// TIA Portal V17 export
// export: Created 2025-03-13T10:29:50.4111857Z, ExportSetting WithDefaults, DisplayName Totally Integrated Automation Portal, DisplayVersion V17 Update 8, DisplayName TIA Portal Openness, DisplayVersion V17 Update 8, DisplayName TIA Portal Version Control Interface, DisplayVersion V17, DisplayName SINAMICS Startdrive Advanced, DisplayVersion V17 SP2, DisplayName SINAMICS Startdrive G110M, G120, G120C, G120D, G120P, G115D, DisplayVersion V17 SP2, DisplayName SINAMICS Startdrive G130, G150, S120, S150, SINAMICS MV, S210, DisplayVersion V17 SP2, DisplayName STEP 7 Professional, DisplayVersion V17 Update 8, DisplayName SINUMERIK ONE STEP 7 Toolbox, DisplayVersion V17 Update 12, DisplayName SINUMERIK 840D sl STEP 7 Toolbox, DisplayVersion V17 Update 12, DisplayName STEP 7 Safety, DisplayVersion V17 Update 6, DisplayName WinCC Advanced, DisplayVersion V17 Update 8
FUNCTION "FC7330_ROBOT_CELL_TO_MACHINE_INTERLOCK" : Void   // FC7330, LAD
{ S7_Optimized_Access := 'FALSE' }
AUTHOR : ETXETAR
VERSION : 1.0
// stored: AutoNumber false, IsIECCheckEnabled false, SetENOAutomatically false, UDAEnableTagReadback false
   VAR_TEMP
      dry_load_side0 : Bool;
      dry_load_side180 : Bool;
      Status_receive : Int;
      QC_FORECAST : Int;
      QC_EXPIRED : Int;
      QC_COUNTS : Int;
      RETVAL_FILL : Int;
      temp0 : Int;
      status_sfc21 : Int;
      RETVAL_FILL_1 : Int;
      ONE : Byte;
      ZERO : Byte;
      retval_sfc21 : Int;
      COUNTS_FOR_ERROR_UNIT_01 : Int;
      COUNTS_FOR_ERROR_UNIT_02 : Int;
      AUX_1_GTRY_SWITCH_OFF : Bool;
      AUX_2_GTRY_SWITCH_OFF : Bool;
      WITH_MANUAL_LOADER : Bool;
      WITH_OUT_MANUAL_LOADER : Bool;
   END_VAR
   VAR CONSTANT
      FC_NUMBER : DInt := 7330;   // FC NUMBER
   END_VAR
   VAR_TEMP   // added for the SCL form of the ladder/FBD networks
      _w1 : Bool;
      _w2 : Bool;
   END_VAR
BEGIN

REGION Network 1: >>>>>>>>>>>>>>>> INTERLOCKS CELL TO MACHINE GENERAL <<<<<<<<<<<<<<<<
END_REGION

REGION Network 2: MEASURING STATION START MEASURING CYCLE
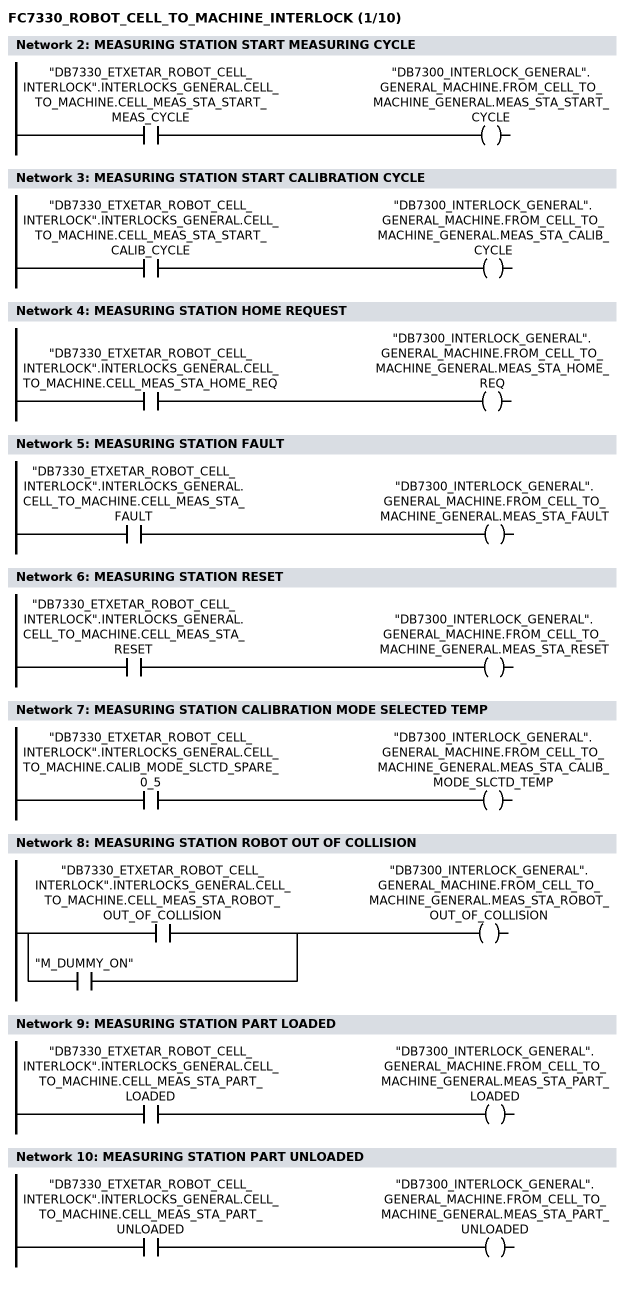
   RUNG wire#powerrail
      Contact( "DB7330_ETXETAR_ROBOT_CELL_INTERLOCK".INTERLOCKS_GENERAL.CELL_TO_MACHINE.CELL_MEAS_STA_START_MEAS_CYCLE )
      Coil( "DB7300_INTERLOCK_GENERAL".GENERAL_MACHINE.FROM_CELL_TO_MACHINE_GENERAL.MEAS_STA_START_CYCLE )
   END_RUNG
   // the same network as SCL:
   "DB7300_INTERLOCK_GENERAL".GENERAL_MACHINE.FROM_CELL_TO_MACHINE_GENERAL.MEAS_STA_START_CYCLE := "DB7330_ETXETAR_ROBOT_CELL_INTERLOCK".INTERLOCKS_GENERAL.CELL_TO_MACHINE.CELL_MEAS_STA_START_MEAS_CYCLE;
END_REGION

REGION Network 3: MEASURING STATION START CALIBRATION CYCLE
   RUNG wire#powerrail
      Contact( "DB7330_ETXETAR_ROBOT_CELL_INTERLOCK".INTERLOCKS_GENERAL.CELL_TO_MACHINE.CELL_MEAS_STA_START_CALIB_CYCLE )
      Coil( "DB7300_INTERLOCK_GENERAL".GENERAL_MACHINE.FROM_CELL_TO_MACHINE_GENERAL.MEAS_STA_CALIB_CYCLE )
   END_RUNG
   // the same network as SCL:
   "DB7300_INTERLOCK_GENERAL".GENERAL_MACHINE.FROM_CELL_TO_MACHINE_GENERAL.MEAS_STA_CALIB_CYCLE := "DB7330_ETXETAR_ROBOT_CELL_INTERLOCK".INTERLOCKS_GENERAL.CELL_TO_MACHINE.CELL_MEAS_STA_START_CALIB_CYCLE;
END_REGION

REGION Network 4: MEASURING STATION HOME REQUEST
   RUNG wire#powerrail
      Contact( "DB7330_ETXETAR_ROBOT_CELL_INTERLOCK".INTERLOCKS_GENERAL.CELL_TO_MACHINE.CELL_MEAS_STA_HOME_REQ )
      Coil( "DB7300_INTERLOCK_GENERAL".GENERAL_MACHINE.FROM_CELL_TO_MACHINE_GENERAL.MEAS_STA_HOME_REQ )
   END_RUNG
   // the same network as SCL:
   "DB7300_INTERLOCK_GENERAL".GENERAL_MACHINE.FROM_CELL_TO_MACHINE_GENERAL.MEAS_STA_HOME_REQ := "DB7330_ETXETAR_ROBOT_CELL_INTERLOCK".INTERLOCKS_GENERAL.CELL_TO_MACHINE.CELL_MEAS_STA_HOME_REQ;
END_REGION

REGION Network 5: MEASURING STATION FAULT
   RUNG wire#powerrail
      Contact( "DB7330_ETXETAR_ROBOT_CELL_INTERLOCK".INTERLOCKS_GENERAL.CELL_TO_MACHINE.CELL_MEAS_STA_FAULT )
      Coil( "DB7300_INTERLOCK_GENERAL".GENERAL_MACHINE.FROM_CELL_TO_MACHINE_GENERAL.MEAS_STA_FAULT )
   END_RUNG
   // the same network as SCL:
   "DB7300_INTERLOCK_GENERAL".GENERAL_MACHINE.FROM_CELL_TO_MACHINE_GENERAL.MEAS_STA_FAULT := "DB7330_ETXETAR_ROBOT_CELL_INTERLOCK".INTERLOCKS_GENERAL.CELL_TO_MACHINE.CELL_MEAS_STA_FAULT;
END_REGION

REGION Network 6: MEASURING STATION RESET
   RUNG wire#powerrail
      Contact( "DB7330_ETXETAR_ROBOT_CELL_INTERLOCK".INTERLOCKS_GENERAL.CELL_TO_MACHINE.CELL_MEAS_STA_RESET )
      Coil( "DB7300_INTERLOCK_GENERAL".GENERAL_MACHINE.FROM_CELL_TO_MACHINE_GENERAL.MEAS_STA_RESET )
   END_RUNG
   // the same network as SCL:
   "DB7300_INTERLOCK_GENERAL".GENERAL_MACHINE.FROM_CELL_TO_MACHINE_GENERAL.MEAS_STA_RESET := "DB7330_ETXETAR_ROBOT_CELL_INTERLOCK".INTERLOCKS_GENERAL.CELL_TO_MACHINE.CELL_MEAS_STA_RESET;
END_REGION

REGION Network 7: MEASURING STATION CALIBRATION MODE SELECTED TEMP
   RUNG wire#powerrail
      Contact( "DB7330_ETXETAR_ROBOT_CELL_INTERLOCK".INTERLOCKS_GENERAL.CELL_TO_MACHINE.CALIB_MODE_SLCTD_SPARE_0_5 )
      Coil( "DB7300_INTERLOCK_GENERAL".GENERAL_MACHINE.FROM_CELL_TO_MACHINE_GENERAL.MEAS_STA_CALIB_MODE_SLCTD_TEMP )
   END_RUNG
   // the same network as SCL:
   "DB7300_INTERLOCK_GENERAL".GENERAL_MACHINE.FROM_CELL_TO_MACHINE_GENERAL.MEAS_STA_CALIB_MODE_SLCTD_TEMP := "DB7330_ETXETAR_ROBOT_CELL_INTERLOCK".INTERLOCKS_GENERAL.CELL_TO_MACHINE.CALIB_MODE_SLCTD_SPARE_0_5;
END_REGION

REGION Network 8: MEASURING STATION ROBOT OUT OF COLLISION
   RUNG wire#powerrail
      Contact( "DB7330_ETXETAR_ROBOT_CELL_INTERLOCK".INTERLOCKS_GENERAL.CELL_TO_MACHINE.CELL_MEAS_STA_ROBOT_OUT_OF_COLLISION )
      wire#w1
      Coil( "DB7300_INTERLOCK_GENERAL".GENERAL_MACHINE.FROM_CELL_TO_MACHINE_GENERAL.MEAS_STA_ROBOT_OUT_OF_COLLISION )
   END_RUNG
   RUNG wire#powerrail
      Contact( "M_DUMMY_ON" )
   END_RUNG wire#w1
   // the same network as SCL:
   "DB7300_INTERLOCK_GENERAL".GENERAL_MACHINE.FROM_CELL_TO_MACHINE_GENERAL.MEAS_STA_ROBOT_OUT_OF_COLLISION := "DB7330_ETXETAR_ROBOT_CELL_INTERLOCK".INTERLOCKS_GENERAL.CELL_TO_MACHINE.CELL_MEAS_STA_ROBOT_OUT_OF_COLLISION OR "M_DUMMY_ON";
END_REGION

REGION Network 9: MEASURING STATION PART LOADED
   RUNG wire#powerrail
      Contact( "DB7330_ETXETAR_ROBOT_CELL_INTERLOCK".INTERLOCKS_GENERAL.CELL_TO_MACHINE.CELL_MEAS_STA_PART_LOADED )
      Coil( "DB7300_INTERLOCK_GENERAL".GENERAL_MACHINE.FROM_CELL_TO_MACHINE_GENERAL.MEAS_STA_PART_LOADED )
   END_RUNG
   // the same network as SCL:
   "DB7300_INTERLOCK_GENERAL".GENERAL_MACHINE.FROM_CELL_TO_MACHINE_GENERAL.MEAS_STA_PART_LOADED := "DB7330_ETXETAR_ROBOT_CELL_INTERLOCK".INTERLOCKS_GENERAL.CELL_TO_MACHINE.CELL_MEAS_STA_PART_LOADED;
END_REGION

REGION Network 10: MEASURING STATION PART UNLOADED
   RUNG wire#powerrail
      Contact( "DB7330_ETXETAR_ROBOT_CELL_INTERLOCK".INTERLOCKS_GENERAL.CELL_TO_MACHINE.CELL_MEAS_STA_PART_UNLOADED )
      Coil( "DB7300_INTERLOCK_GENERAL".GENERAL_MACHINE.FROM_CELL_TO_MACHINE_GENERAL.MEAS_STA_PART_UNLOADED )
   END_RUNG
   // the same network as SCL:
   "DB7300_INTERLOCK_GENERAL".GENERAL_MACHINE.FROM_CELL_TO_MACHINE_GENERAL.MEAS_STA_PART_UNLOADED := "DB7330_ETXETAR_ROBOT_CELL_INTERLOCK".INTERLOCKS_GENERAL.CELL_TO_MACHINE.CELL_MEAS_STA_PART_UNLOADED;
END_REGION

REGION Network 11: CELL COOLING DEGRADED MODE
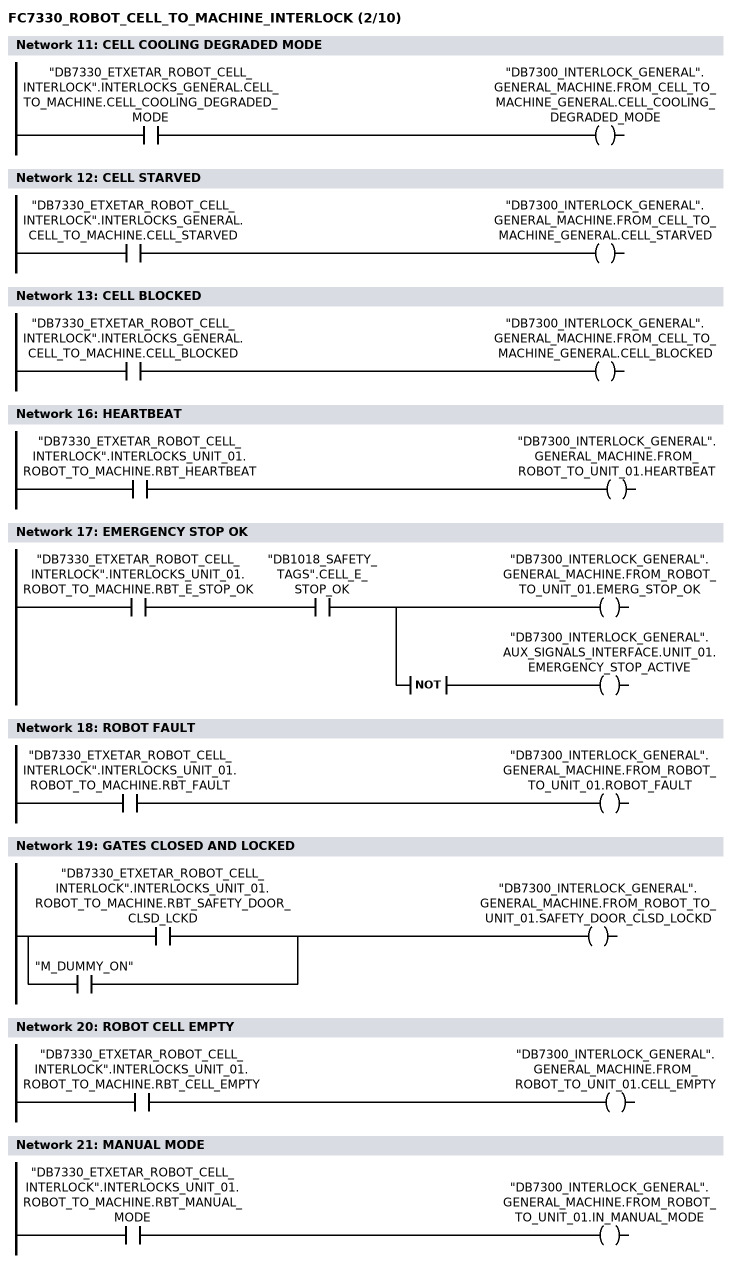
   RUNG wire#powerrail
      Contact( "DB7330_ETXETAR_ROBOT_CELL_INTERLOCK".INTERLOCKS_GENERAL.CELL_TO_MACHINE.CELL_COOLING_DEGRADED_MODE )
      Coil( "DB7300_INTERLOCK_GENERAL".GENERAL_MACHINE.FROM_CELL_TO_MACHINE_GENERAL.CELL_COOLING_DEGRADED_MODE )
   END_RUNG
   // the same network as SCL:
   "DB7300_INTERLOCK_GENERAL".GENERAL_MACHINE.FROM_CELL_TO_MACHINE_GENERAL.CELL_COOLING_DEGRADED_MODE := "DB7330_ETXETAR_ROBOT_CELL_INTERLOCK".INTERLOCKS_GENERAL.CELL_TO_MACHINE.CELL_COOLING_DEGRADED_MODE;
END_REGION

REGION Network 12: CELL STARVED
   RUNG wire#powerrail
      Contact( "DB7330_ETXETAR_ROBOT_CELL_INTERLOCK".INTERLOCKS_GENERAL.CELL_TO_MACHINE.CELL_STARVED )
      Coil( "DB7300_INTERLOCK_GENERAL".GENERAL_MACHINE.FROM_CELL_TO_MACHINE_GENERAL.CELL_STARVED )
   END_RUNG
   // the same network as SCL:
   "DB7300_INTERLOCK_GENERAL".GENERAL_MACHINE.FROM_CELL_TO_MACHINE_GENERAL.CELL_STARVED := "DB7330_ETXETAR_ROBOT_CELL_INTERLOCK".INTERLOCKS_GENERAL.CELL_TO_MACHINE.CELL_STARVED;
END_REGION

REGION Network 13: CELL BLOCKED
   RUNG wire#powerrail
      Contact( "DB7330_ETXETAR_ROBOT_CELL_INTERLOCK".INTERLOCKS_GENERAL.CELL_TO_MACHINE.CELL_BLOCKED )
      Coil( "DB7300_INTERLOCK_GENERAL".GENERAL_MACHINE.FROM_CELL_TO_MACHINE_GENERAL.CELL_BLOCKED )
   END_RUNG
   // the same network as SCL:
   "DB7300_INTERLOCK_GENERAL".GENERAL_MACHINE.FROM_CELL_TO_MACHINE_GENERAL.CELL_BLOCKED := "DB7330_ETXETAR_ROBOT_CELL_INTERLOCK".INTERLOCKS_GENERAL.CELL_TO_MACHINE.CELL_BLOCKED;
END_REGION

REGION Network 15: >>>>>>>>>>>>>>>> INTERLOCKS ROBOT TO MACHINE UNIT 01 <<<<<<<<<<<<<<<<
END_REGION

REGION Network 16: HEARTBEAT
   RUNG wire#powerrail
      Contact( "DB7330_ETXETAR_ROBOT_CELL_INTERLOCK".INTERLOCKS_UNIT_01.ROBOT_TO_MACHINE.RBT_HEARTBEAT )
      Coil( "DB7300_INTERLOCK_GENERAL".GENERAL_MACHINE.FROM_ROBOT_TO_UNIT_01.HEARTBEAT )
   END_RUNG
   // the same network as SCL:
   "DB7300_INTERLOCK_GENERAL".GENERAL_MACHINE.FROM_ROBOT_TO_UNIT_01.HEARTBEAT := "DB7330_ETXETAR_ROBOT_CELL_INTERLOCK".INTERLOCKS_UNIT_01.ROBOT_TO_MACHINE.RBT_HEARTBEAT;
END_REGION

REGION Network 17: EMERGENCY STOP OK
   RUNG wire#powerrail
      Contact( "DB7330_ETXETAR_ROBOT_CELL_INTERLOCK".INTERLOCKS_UNIT_01.ROBOT_TO_MACHINE.RBT_E_STOP_OK )
      Contact( "DB1018_SAFETY_TAGS".CELL_E_STOP_OK )
      wire#w1
      Coil( "DB7300_INTERLOCK_GENERAL".GENERAL_MACHINE.FROM_ROBOT_TO_UNIT_01.EMERG_STOP_OK )
   END_RUNG
   RUNG wire#w1
      Not()
      Coil( "DB7300_INTERLOCK_GENERAL".AUX_SIGNALS_INTERFACE.UNIT_01.EMERGENCY_STOP_ACTIVE )
   END_RUNG
   // the same network as SCL:
   "DB7300_INTERLOCK_GENERAL".GENERAL_MACHINE.FROM_ROBOT_TO_UNIT_01.EMERG_STOP_OK := "DB7330_ETXETAR_ROBOT_CELL_INTERLOCK".INTERLOCKS_UNIT_01.ROBOT_TO_MACHINE.RBT_E_STOP_OK AND "DB1018_SAFETY_TAGS".CELL_E_STOP_OK;
   "DB7300_INTERLOCK_GENERAL".AUX_SIGNALS_INTERFACE.UNIT_01.EMERGENCY_STOP_ACTIVE := NOT "DB7300_INTERLOCK_GENERAL".GENERAL_MACHINE.FROM_ROBOT_TO_UNIT_01.EMERG_STOP_OK;
END_REGION

REGION Network 18: ROBOT FAULT
   RUNG wire#powerrail
      Contact( "DB7330_ETXETAR_ROBOT_CELL_INTERLOCK".INTERLOCKS_UNIT_01.ROBOT_TO_MACHINE.RBT_FAULT )
      Coil( "DB7300_INTERLOCK_GENERAL".GENERAL_MACHINE.FROM_ROBOT_TO_UNIT_01.ROBOT_FAULT )
   END_RUNG
   // the same network as SCL:
   "DB7300_INTERLOCK_GENERAL".GENERAL_MACHINE.FROM_ROBOT_TO_UNIT_01.ROBOT_FAULT := "DB7330_ETXETAR_ROBOT_CELL_INTERLOCK".INTERLOCKS_UNIT_01.ROBOT_TO_MACHINE.RBT_FAULT;
END_REGION

REGION Network 19: GATES CLOSED AND LOCKED
   RUNG wire#powerrail
      Contact( "DB7330_ETXETAR_ROBOT_CELL_INTERLOCK".INTERLOCKS_UNIT_01.ROBOT_TO_MACHINE.RBT_SAFETY_DOOR_CLSD_LCKD )
      wire#w1
      Coil( "DB7300_INTERLOCK_GENERAL".GENERAL_MACHINE.FROM_ROBOT_TO_UNIT_01.SAFETY_DOOR_CLSD_LOCKD )
   END_RUNG
   RUNG wire#powerrail
      Contact( "M_DUMMY_ON" )
   END_RUNG wire#w1
   // the same network as SCL:
   "DB7300_INTERLOCK_GENERAL".GENERAL_MACHINE.FROM_ROBOT_TO_UNIT_01.SAFETY_DOOR_CLSD_LOCKD := "DB7330_ETXETAR_ROBOT_CELL_INTERLOCK".INTERLOCKS_UNIT_01.ROBOT_TO_MACHINE.RBT_SAFETY_DOOR_CLSD_LCKD OR "M_DUMMY_ON";
END_REGION

REGION Network 20: ROBOT CELL EMPTY
   RUNG wire#powerrail
      Contact( "DB7330_ETXETAR_ROBOT_CELL_INTERLOCK".INTERLOCKS_UNIT_01.ROBOT_TO_MACHINE.RBT_CELL_EMPTY )
      Coil( "DB7300_INTERLOCK_GENERAL".GENERAL_MACHINE.FROM_ROBOT_TO_UNIT_01.CELL_EMPTY )
   END_RUNG
   // the same network as SCL:
   "DB7300_INTERLOCK_GENERAL".GENERAL_MACHINE.FROM_ROBOT_TO_UNIT_01.CELL_EMPTY := "DB7330_ETXETAR_ROBOT_CELL_INTERLOCK".INTERLOCKS_UNIT_01.ROBOT_TO_MACHINE.RBT_CELL_EMPTY;
END_REGION

REGION Network 21: MANUAL MODE
   RUNG wire#powerrail
      Contact( "DB7330_ETXETAR_ROBOT_CELL_INTERLOCK".INTERLOCKS_UNIT_01.ROBOT_TO_MACHINE.RBT_MANUAL_MODE )
      Coil( "DB7300_INTERLOCK_GENERAL".GENERAL_MACHINE.FROM_ROBOT_TO_UNIT_01.IN_MANUAL_MODE )
   END_RUNG
   // the same network as SCL:
   "DB7300_INTERLOCK_GENERAL".GENERAL_MACHINE.FROM_ROBOT_TO_UNIT_01.IN_MANUAL_MODE := "DB7330_ETXETAR_ROBOT_CELL_INTERLOCK".INTERLOCKS_UNIT_01.ROBOT_TO_MACHINE.RBT_MANUAL_MODE;
END_REGION

REGION Network 22: AUTO MODE
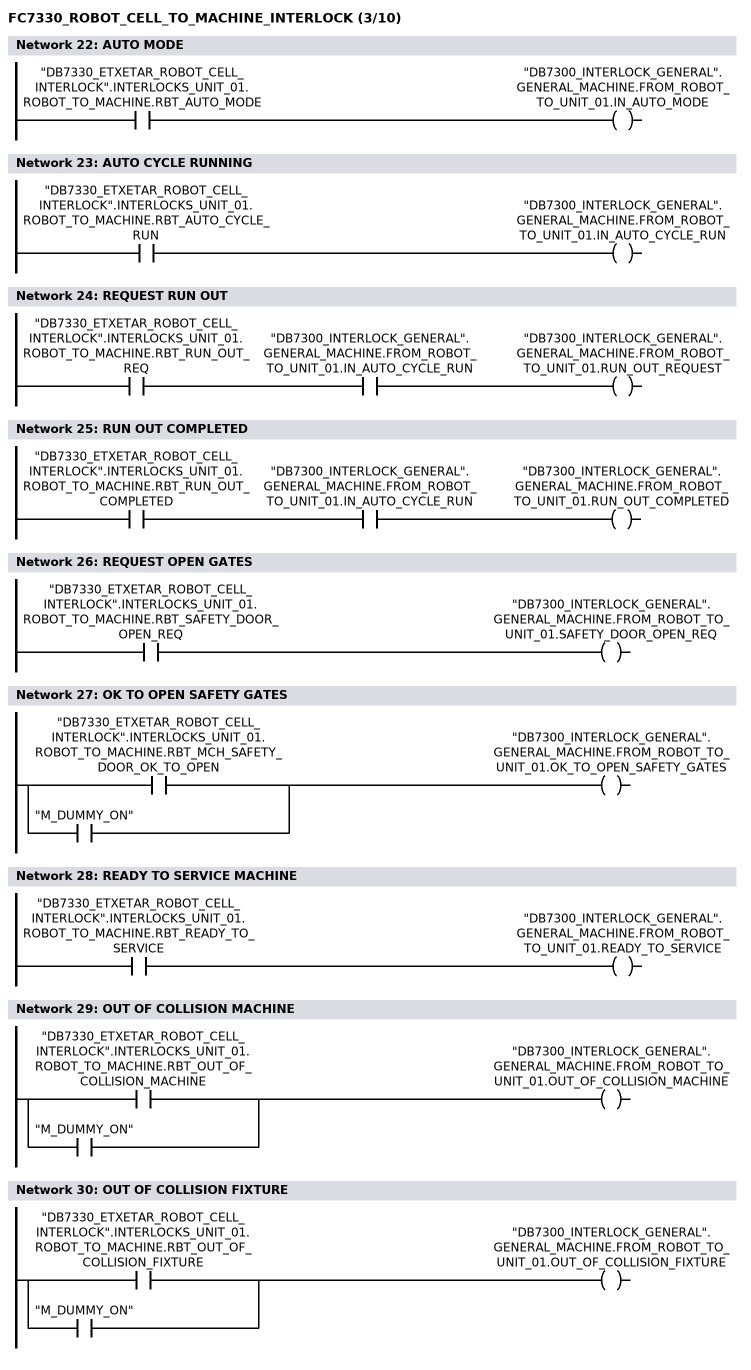
   RUNG wire#powerrail
      Contact( "DB7330_ETXETAR_ROBOT_CELL_INTERLOCK".INTERLOCKS_UNIT_01.ROBOT_TO_MACHINE.RBT_AUTO_MODE )
      Coil( "DB7300_INTERLOCK_GENERAL".GENERAL_MACHINE.FROM_ROBOT_TO_UNIT_01.IN_AUTO_MODE )
   END_RUNG
   // the same network as SCL:
   "DB7300_INTERLOCK_GENERAL".GENERAL_MACHINE.FROM_ROBOT_TO_UNIT_01.IN_AUTO_MODE := "DB7330_ETXETAR_ROBOT_CELL_INTERLOCK".INTERLOCKS_UNIT_01.ROBOT_TO_MACHINE.RBT_AUTO_MODE;
END_REGION

REGION Network 23: AUTO CYCLE RUNNING
   RUNG wire#powerrail
      Contact( "DB7330_ETXETAR_ROBOT_CELL_INTERLOCK".INTERLOCKS_UNIT_01.ROBOT_TO_MACHINE.RBT_AUTO_CYCLE_RUN )
      Coil( "DB7300_INTERLOCK_GENERAL".GENERAL_MACHINE.FROM_ROBOT_TO_UNIT_01.IN_AUTO_CYCLE_RUN )
   END_RUNG
   // the same network as SCL:
   "DB7300_INTERLOCK_GENERAL".GENERAL_MACHINE.FROM_ROBOT_TO_UNIT_01.IN_AUTO_CYCLE_RUN := "DB7330_ETXETAR_ROBOT_CELL_INTERLOCK".INTERLOCKS_UNIT_01.ROBOT_TO_MACHINE.RBT_AUTO_CYCLE_RUN;
END_REGION

REGION Network 24: REQUEST RUN OUT
   RUNG wire#powerrail
      Contact( "DB7330_ETXETAR_ROBOT_CELL_INTERLOCK".INTERLOCKS_UNIT_01.ROBOT_TO_MACHINE.RBT_RUN_OUT_REQ )
      Contact( "DB7300_INTERLOCK_GENERAL".GENERAL_MACHINE.FROM_ROBOT_TO_UNIT_01.IN_AUTO_CYCLE_RUN )
      Coil( "DB7300_INTERLOCK_GENERAL".GENERAL_MACHINE.FROM_ROBOT_TO_UNIT_01.RUN_OUT_REQUEST )
   END_RUNG
   // the same network as SCL:
   "DB7300_INTERLOCK_GENERAL".GENERAL_MACHINE.FROM_ROBOT_TO_UNIT_01.RUN_OUT_REQUEST := "DB7330_ETXETAR_ROBOT_CELL_INTERLOCK".INTERLOCKS_UNIT_01.ROBOT_TO_MACHINE.RBT_RUN_OUT_REQ AND "DB7300_INTERLOCK_GENERAL".GENERAL_MACHINE.FROM_ROBOT_TO_UNIT_01.IN_AUTO_CYCLE_RUN;
END_REGION

REGION Network 25: RUN OUT COMPLETED
   RUNG wire#powerrail
      Contact( "DB7330_ETXETAR_ROBOT_CELL_INTERLOCK".INTERLOCKS_UNIT_01.ROBOT_TO_MACHINE.RBT_RUN_OUT_COMPLETED )
      Contact( "DB7300_INTERLOCK_GENERAL".GENERAL_MACHINE.FROM_ROBOT_TO_UNIT_01.IN_AUTO_CYCLE_RUN )
      Coil( "DB7300_INTERLOCK_GENERAL".GENERAL_MACHINE.FROM_ROBOT_TO_UNIT_01.RUN_OUT_COMPLETED )
   END_RUNG
   // the same network as SCL:
   "DB7300_INTERLOCK_GENERAL".GENERAL_MACHINE.FROM_ROBOT_TO_UNIT_01.RUN_OUT_COMPLETED := "DB7330_ETXETAR_ROBOT_CELL_INTERLOCK".INTERLOCKS_UNIT_01.ROBOT_TO_MACHINE.RBT_RUN_OUT_COMPLETED AND "DB7300_INTERLOCK_GENERAL".GENERAL_MACHINE.FROM_ROBOT_TO_UNIT_01.IN_AUTO_CYCLE_RUN;
END_REGION

REGION Network 26: REQUEST OPEN GATES
   RUNG wire#powerrail
      Contact( "DB7330_ETXETAR_ROBOT_CELL_INTERLOCK".INTERLOCKS_UNIT_01.ROBOT_TO_MACHINE.RBT_SAFETY_DOOR_OPEN_REQ )
      Coil( "DB7300_INTERLOCK_GENERAL".GENERAL_MACHINE.FROM_ROBOT_TO_UNIT_01.SAFETY_DOOR_OPEN_REQ )
   END_RUNG
   // the same network as SCL:
   "DB7300_INTERLOCK_GENERAL".GENERAL_MACHINE.FROM_ROBOT_TO_UNIT_01.SAFETY_DOOR_OPEN_REQ := "DB7330_ETXETAR_ROBOT_CELL_INTERLOCK".INTERLOCKS_UNIT_01.ROBOT_TO_MACHINE.RBT_SAFETY_DOOR_OPEN_REQ;
END_REGION

REGION Network 27: OK TO OPEN SAFETY GATES
   RUNG wire#powerrail
      Contact( "DB7330_ETXETAR_ROBOT_CELL_INTERLOCK".INTERLOCKS_UNIT_01.ROBOT_TO_MACHINE.RBT_MCH_SAFETY_DOOR_OK_TO_OPEN )
      wire#w1
      Coil( "DB7300_INTERLOCK_GENERAL".GENERAL_MACHINE.FROM_ROBOT_TO_UNIT_01.OK_TO_OPEN_SAFETY_GATES )
   END_RUNG
   RUNG wire#powerrail
      Contact( "M_DUMMY_ON" )
   END_RUNG wire#w1
   // the same network as SCL:
   "DB7300_INTERLOCK_GENERAL".GENERAL_MACHINE.FROM_ROBOT_TO_UNIT_01.OK_TO_OPEN_SAFETY_GATES := "DB7330_ETXETAR_ROBOT_CELL_INTERLOCK".INTERLOCKS_UNIT_01.ROBOT_TO_MACHINE.RBT_MCH_SAFETY_DOOR_OK_TO_OPEN OR "M_DUMMY_ON";
END_REGION

REGION Network 28: READY TO SERVICE MACHINE
   RUNG wire#powerrail
      Contact( "DB7330_ETXETAR_ROBOT_CELL_INTERLOCK".INTERLOCKS_UNIT_01.ROBOT_TO_MACHINE.RBT_READY_TO_SERVICE )
      Coil( "DB7300_INTERLOCK_GENERAL".GENERAL_MACHINE.FROM_ROBOT_TO_UNIT_01.READY_TO_SERVICE )
   END_RUNG
   // the same network as SCL:
   "DB7300_INTERLOCK_GENERAL".GENERAL_MACHINE.FROM_ROBOT_TO_UNIT_01.READY_TO_SERVICE := "DB7330_ETXETAR_ROBOT_CELL_INTERLOCK".INTERLOCKS_UNIT_01.ROBOT_TO_MACHINE.RBT_READY_TO_SERVICE;
END_REGION

REGION Network 29: OUT OF COLLISION MACHINE
   RUNG wire#powerrail
      Contact( "DB7330_ETXETAR_ROBOT_CELL_INTERLOCK".INTERLOCKS_UNIT_01.ROBOT_TO_MACHINE.RBT_OUT_OF_COLLISION_MACHINE )
      wire#w1
      Coil( "DB7300_INTERLOCK_GENERAL".GENERAL_MACHINE.FROM_ROBOT_TO_UNIT_01.OUT_OF_COLLISION_MACHINE )
   END_RUNG
   RUNG wire#powerrail
      Contact( "M_DUMMY_ON" )
   END_RUNG wire#w1
   // the same network as SCL:
   "DB7300_INTERLOCK_GENERAL".GENERAL_MACHINE.FROM_ROBOT_TO_UNIT_01.OUT_OF_COLLISION_MACHINE := "DB7330_ETXETAR_ROBOT_CELL_INTERLOCK".INTERLOCKS_UNIT_01.ROBOT_TO_MACHINE.RBT_OUT_OF_COLLISION_MACHINE OR "M_DUMMY_ON";
END_REGION

REGION Network 30: OUT OF COLLISION FIXTURE
   RUNG wire#powerrail
      Contact( "DB7330_ETXETAR_ROBOT_CELL_INTERLOCK".INTERLOCKS_UNIT_01.ROBOT_TO_MACHINE.RBT_OUT_OF_COLLISION_FIXTURE )
      wire#w1
      Coil( "DB7300_INTERLOCK_GENERAL".GENERAL_MACHINE.FROM_ROBOT_TO_UNIT_01.OUT_OF_COLLISION_FIXTURE )
   END_RUNG
   RUNG wire#powerrail
      Contact( "M_DUMMY_ON" )
   END_RUNG wire#w1
   // the same network as SCL:
   "DB7300_INTERLOCK_GENERAL".GENERAL_MACHINE.FROM_ROBOT_TO_UNIT_01.OUT_OF_COLLISION_FIXTURE := "DB7330_ETXETAR_ROBOT_CELL_INTERLOCK".INTERLOCKS_UNIT_01.ROBOT_TO_MACHINE.RBT_OUT_OF_COLLISION_FIXTURE OR "M_DUMMY_ON";
END_REGION

REGION Network 31: PART ENABLED
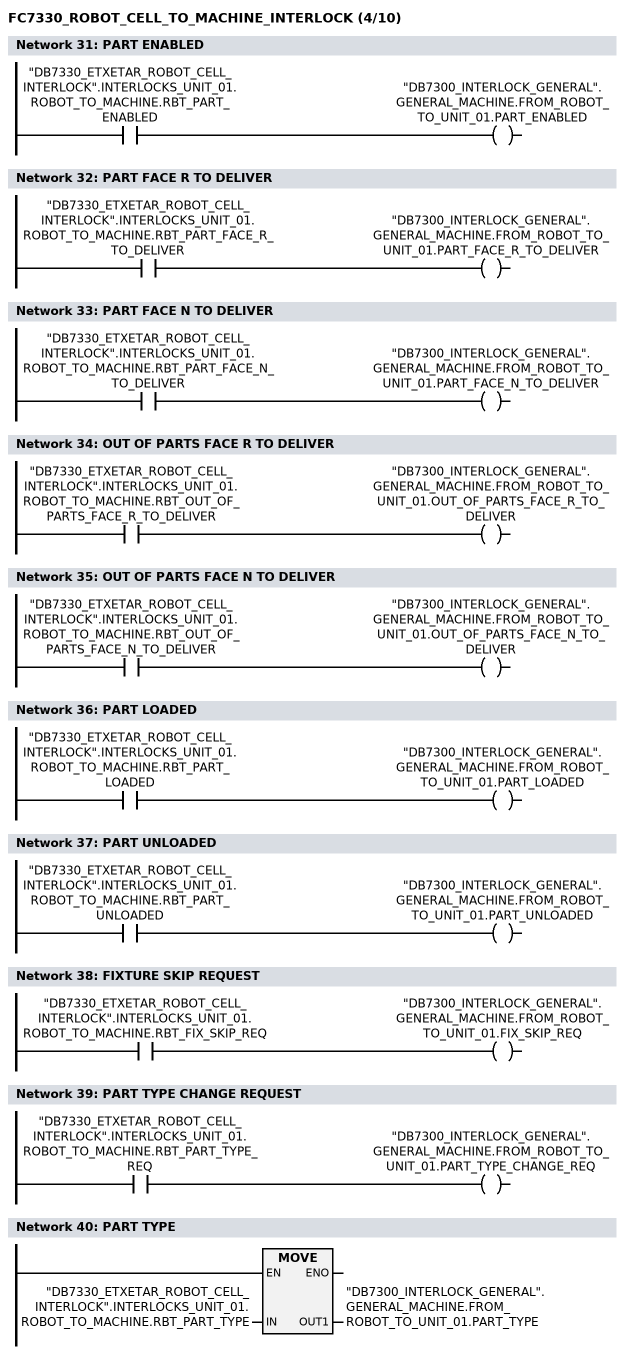
   RUNG wire#powerrail
      Contact( "DB7330_ETXETAR_ROBOT_CELL_INTERLOCK".INTERLOCKS_UNIT_01.ROBOT_TO_MACHINE.RBT_PART_ENABLED )
      Coil( "DB7300_INTERLOCK_GENERAL".GENERAL_MACHINE.FROM_ROBOT_TO_UNIT_01.PART_ENABLED )
   END_RUNG
   // the same network as SCL:
   "DB7300_INTERLOCK_GENERAL".GENERAL_MACHINE.FROM_ROBOT_TO_UNIT_01.PART_ENABLED := "DB7330_ETXETAR_ROBOT_CELL_INTERLOCK".INTERLOCKS_UNIT_01.ROBOT_TO_MACHINE.RBT_PART_ENABLED;
END_REGION

REGION Network 32: PART FACE R TO DELIVER
   RUNG wire#powerrail
      Contact( "DB7330_ETXETAR_ROBOT_CELL_INTERLOCK".INTERLOCKS_UNIT_01.ROBOT_TO_MACHINE.RBT_PART_FACE_R_TO_DELIVER )
      Coil( "DB7300_INTERLOCK_GENERAL".GENERAL_MACHINE.FROM_ROBOT_TO_UNIT_01.PART_FACE_R_TO_DELIVER )
   END_RUNG
   // the same network as SCL:
   "DB7300_INTERLOCK_GENERAL".GENERAL_MACHINE.FROM_ROBOT_TO_UNIT_01.PART_FACE_R_TO_DELIVER := "DB7330_ETXETAR_ROBOT_CELL_INTERLOCK".INTERLOCKS_UNIT_01.ROBOT_TO_MACHINE.RBT_PART_FACE_R_TO_DELIVER;
END_REGION

REGION Network 33: PART FACE N TO DELIVER
   RUNG wire#powerrail
      Contact( "DB7330_ETXETAR_ROBOT_CELL_INTERLOCK".INTERLOCKS_UNIT_01.ROBOT_TO_MACHINE.RBT_PART_FACE_N_TO_DELIVER )
      Coil( "DB7300_INTERLOCK_GENERAL".GENERAL_MACHINE.FROM_ROBOT_TO_UNIT_01.PART_FACE_N_TO_DELIVER )
   END_RUNG
   // the same network as SCL:
   "DB7300_INTERLOCK_GENERAL".GENERAL_MACHINE.FROM_ROBOT_TO_UNIT_01.PART_FACE_N_TO_DELIVER := "DB7330_ETXETAR_ROBOT_CELL_INTERLOCK".INTERLOCKS_UNIT_01.ROBOT_TO_MACHINE.RBT_PART_FACE_N_TO_DELIVER;
END_REGION

REGION Network 34: OUT OF PARTS FACE R TO DELIVER
   RUNG wire#powerrail
      Contact( "DB7330_ETXETAR_ROBOT_CELL_INTERLOCK".INTERLOCKS_UNIT_01.ROBOT_TO_MACHINE.RBT_OUT_OF_PARTS_FACE_R_TO_DELIVER )
      Coil( "DB7300_INTERLOCK_GENERAL".GENERAL_MACHINE.FROM_ROBOT_TO_UNIT_01.OUT_OF_PARTS_FACE_R_TO_DELIVER )
   END_RUNG
   // the same network as SCL:
   "DB7300_INTERLOCK_GENERAL".GENERAL_MACHINE.FROM_ROBOT_TO_UNIT_01.OUT_OF_PARTS_FACE_R_TO_DELIVER := "DB7330_ETXETAR_ROBOT_CELL_INTERLOCK".INTERLOCKS_UNIT_01.ROBOT_TO_MACHINE.RBT_OUT_OF_PARTS_FACE_R_TO_DELIVER;
END_REGION

REGION Network 35: OUT OF PARTS FACE N TO DELIVER
   RUNG wire#powerrail
      Contact( "DB7330_ETXETAR_ROBOT_CELL_INTERLOCK".INTERLOCKS_UNIT_01.ROBOT_TO_MACHINE.RBT_OUT_OF_PARTS_FACE_N_TO_DELIVER )
      Coil( "DB7300_INTERLOCK_GENERAL".GENERAL_MACHINE.FROM_ROBOT_TO_UNIT_01.OUT_OF_PARTS_FACE_N_TO_DELIVER )
   END_RUNG
   // the same network as SCL:
   "DB7300_INTERLOCK_GENERAL".GENERAL_MACHINE.FROM_ROBOT_TO_UNIT_01.OUT_OF_PARTS_FACE_N_TO_DELIVER := "DB7330_ETXETAR_ROBOT_CELL_INTERLOCK".INTERLOCKS_UNIT_01.ROBOT_TO_MACHINE.RBT_OUT_OF_PARTS_FACE_N_TO_DELIVER;
END_REGION

REGION Network 36: PART LOADED
   RUNG wire#powerrail
      Contact( "DB7330_ETXETAR_ROBOT_CELL_INTERLOCK".INTERLOCKS_UNIT_01.ROBOT_TO_MACHINE.RBT_PART_LOADED )
      Coil( "DB7300_INTERLOCK_GENERAL".GENERAL_MACHINE.FROM_ROBOT_TO_UNIT_01.PART_LOADED )
   END_RUNG
   // the same network as SCL:
   "DB7300_INTERLOCK_GENERAL".GENERAL_MACHINE.FROM_ROBOT_TO_UNIT_01.PART_LOADED := "DB7330_ETXETAR_ROBOT_CELL_INTERLOCK".INTERLOCKS_UNIT_01.ROBOT_TO_MACHINE.RBT_PART_LOADED;
END_REGION

REGION Network 37: PART UNLOADED
   RUNG wire#powerrail
      Contact( "DB7330_ETXETAR_ROBOT_CELL_INTERLOCK".INTERLOCKS_UNIT_01.ROBOT_TO_MACHINE.RBT_PART_UNLOADED )
      Coil( "DB7300_INTERLOCK_GENERAL".GENERAL_MACHINE.FROM_ROBOT_TO_UNIT_01.PART_UNLOADED )
   END_RUNG
   // the same network as SCL:
   "DB7300_INTERLOCK_GENERAL".GENERAL_MACHINE.FROM_ROBOT_TO_UNIT_01.PART_UNLOADED := "DB7330_ETXETAR_ROBOT_CELL_INTERLOCK".INTERLOCKS_UNIT_01.ROBOT_TO_MACHINE.RBT_PART_UNLOADED;
END_REGION

REGION Network 38: FIXTURE SKIP REQUEST
   RUNG wire#powerrail
      Contact( "DB7330_ETXETAR_ROBOT_CELL_INTERLOCK".INTERLOCKS_UNIT_01.ROBOT_TO_MACHINE.RBT_FIX_SKIP_REQ )
      Coil( "DB7300_INTERLOCK_GENERAL".GENERAL_MACHINE.FROM_ROBOT_TO_UNIT_01.FIX_SKIP_REQ )
   END_RUNG
   // the same network as SCL:
   "DB7300_INTERLOCK_GENERAL".GENERAL_MACHINE.FROM_ROBOT_TO_UNIT_01.FIX_SKIP_REQ := "DB7330_ETXETAR_ROBOT_CELL_INTERLOCK".INTERLOCKS_UNIT_01.ROBOT_TO_MACHINE.RBT_FIX_SKIP_REQ;
END_REGION

REGION Network 39: PART TYPE CHANGE REQUEST
   RUNG wire#powerrail
      Contact( "DB7330_ETXETAR_ROBOT_CELL_INTERLOCK".INTERLOCKS_UNIT_01.ROBOT_TO_MACHINE.RBT_PART_TYPE_REQ )
      Coil( "DB7300_INTERLOCK_GENERAL".GENERAL_MACHINE.FROM_ROBOT_TO_UNIT_01.PART_TYPE_CHANGE_REQ )
   END_RUNG
   // the same network as SCL:
   "DB7300_INTERLOCK_GENERAL".GENERAL_MACHINE.FROM_ROBOT_TO_UNIT_01.PART_TYPE_CHANGE_REQ := "DB7330_ETXETAR_ROBOT_CELL_INTERLOCK".INTERLOCKS_UNIT_01.ROBOT_TO_MACHINE.RBT_PART_TYPE_REQ;
END_REGION

REGION Network 40: PART TYPE
   RUNG wire#powerrail
      { S7_GenerateENO := "TRUE" } Move(in := "DB7330_ETXETAR_ROBOT_CELL_INTERLOCK".INTERLOCKS_UNIT_01.ROBOT_TO_MACHINE.RBT_PART_TYPE, out1 => "DB7300_INTERLOCK_GENERAL".GENERAL_MACHINE.FROM_ROBOT_TO_UNIT_01.PART_TYPE)
   END_RUNG
   // the same network as SCL:
   "DB7300_INTERLOCK_GENERAL".GENERAL_MACHINE.FROM_ROBOT_TO_UNIT_01.PART_TYPE := "DB7330_ETXETAR_ROBOT_CELL_INTERLOCK".INTERLOCKS_UNIT_01.ROBOT_TO_MACHINE.RBT_PART_TYPE;
END_REGION

REGION Network 41: HEARTBEAT COMMUNICATION AUX ALARM
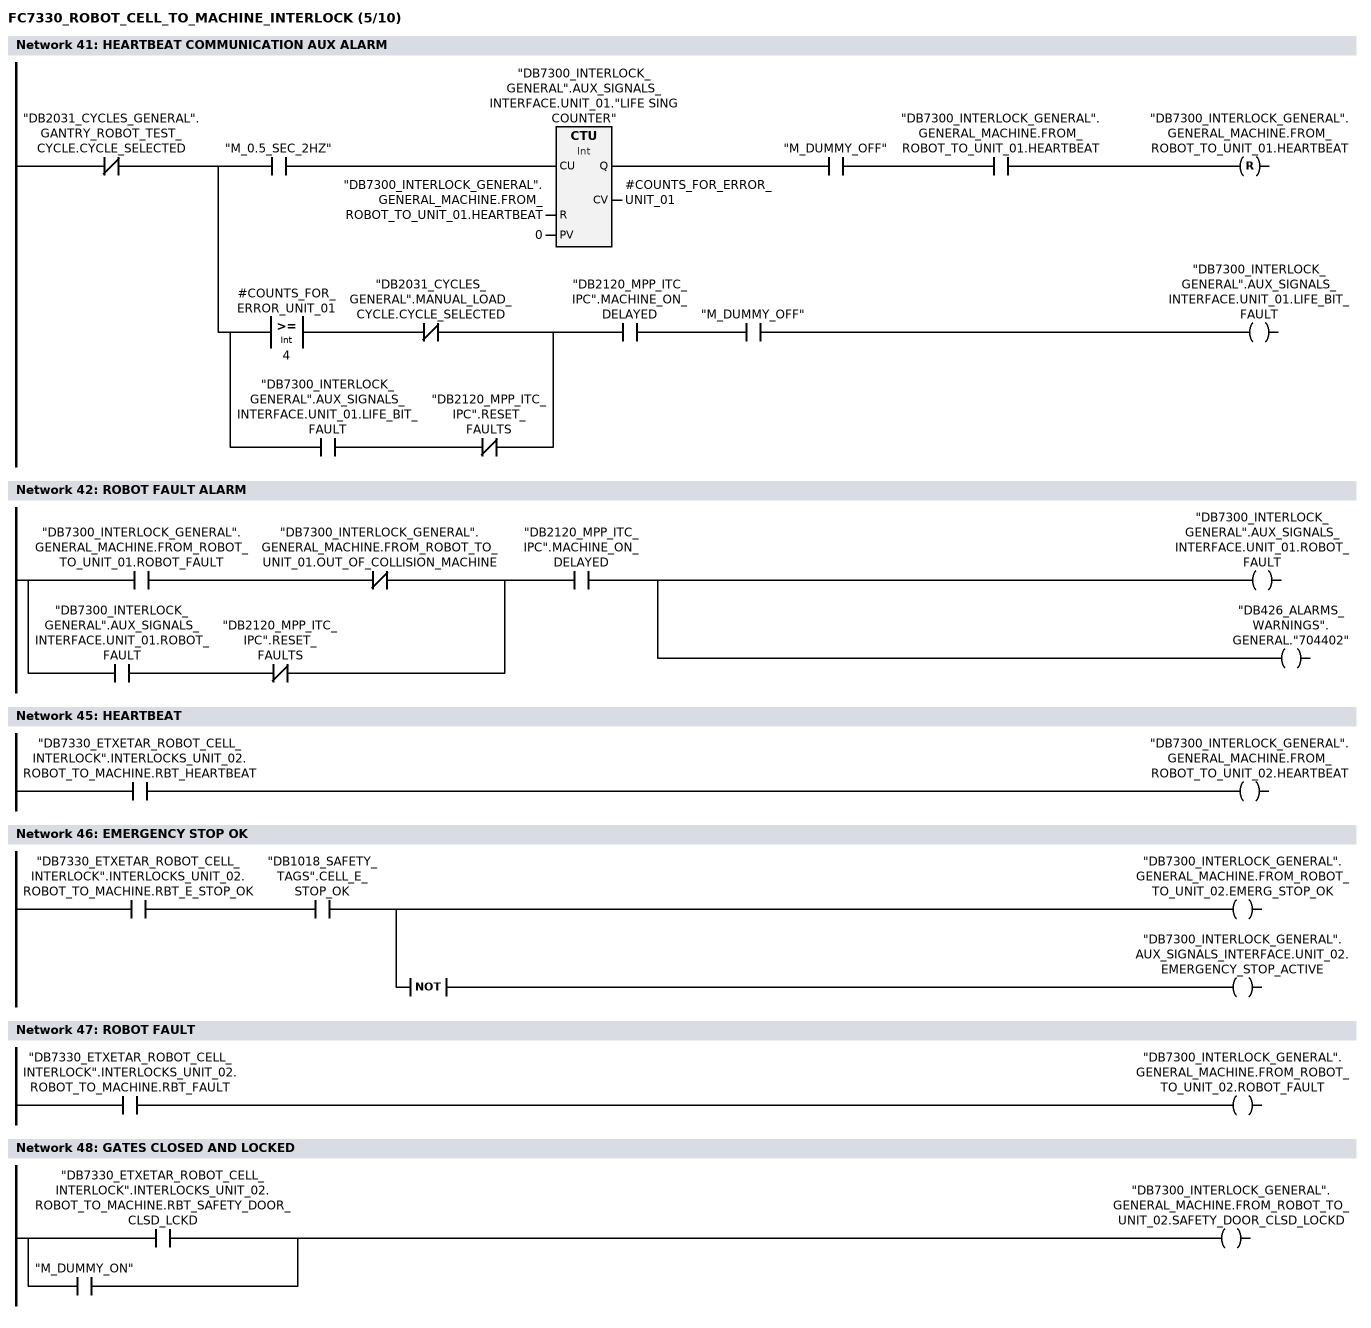
   RUNG wire#powerrail
      I_Contact( "DB2031_CYCLES_GENERAL".GANTRY_ROBOT_TEST_CYCLE.CYCLE_SELECTED )
      wire#w1
      Contact( "M_0.5_SEC_2HZ" )
      { S7_Templates := "value_type := Int" } "DB7300_INTERLOCK_GENERAL".AUX_SIGNALS_INTERFACE.UNIT_01."LIFE SING COUNTER".CTU(r := "DB7300_INTERLOCK_GENERAL".GENERAL_MACHINE.FROM_ROBOT_TO_UNIT_01.HEARTBEAT, pv := 0, cv => #COUNTS_FOR_ERROR_UNIT_01)
      Contact( "M_DUMMY_OFF" )
      Contact( "DB7300_INTERLOCK_GENERAL".GENERAL_MACHINE.FROM_ROBOT_TO_UNIT_01.HEARTBEAT )
      R_Coil( "DB7300_INTERLOCK_GENERAL".GENERAL_MACHINE.FROM_ROBOT_TO_UNIT_01.HEARTBEAT )
   END_RUNG
   RUNG wire#w1
      { S7_Templates := "SrcType := Int" } GE_Contact(in1 := #COUNTS_FOR_ERROR_UNIT_01, in2 := 4)
      I_Contact( "DB2031_CYCLES_GENERAL".MANUAL_LOAD_CYCLE.CYCLE_SELECTED )
      wire#w2
      Contact( "DB2120_MPP_ITC_IPC".MACHINE_ON_DELAYED )
      Contact( "M_DUMMY_OFF" )
      Coil( "DB7300_INTERLOCK_GENERAL".AUX_SIGNALS_INTERFACE.UNIT_01.LIFE_BIT_FAULT )
   END_RUNG
   RUNG wire#w1
      Contact( "DB7300_INTERLOCK_GENERAL".AUX_SIGNALS_INTERFACE.UNIT_01.LIFE_BIT_FAULT )
      I_Contact( "DB2120_MPP_ITC_IPC".RESET_FAULTS )
   END_RUNG wire#w2
   // the same network as SCL:
   #_w1 := NOT "DB2031_CYCLES_GENERAL".GANTRY_ROBOT_TEST_CYCLE.CYCLE_SELECTED;
   "DB7300_INTERLOCK_GENERAL".AUX_SIGNALS_INTERFACE.UNIT_01."LIFE SING COUNTER".CTU(CU := #_w1 AND "M_0.5_SEC_2HZ",
                           R := "DB7300_INTERLOCK_GENERAL".GENERAL_MACHINE.FROM_ROBOT_TO_UNIT_01.HEARTBEAT,
                           PV := 0,
                           CV => #COUNTS_FOR_ERROR_UNIT_01);
   IF "DB7300_INTERLOCK_GENERAL".AUX_SIGNALS_INTERFACE.UNIT_01."LIFE SING COUNTER".Q AND "M_DUMMY_OFF" AND "DB7300_INTERLOCK_GENERAL".GENERAL_MACHINE.FROM_ROBOT_TO_UNIT_01.HEARTBEAT THEN
       "DB7300_INTERLOCK_GENERAL".GENERAL_MACHINE.FROM_ROBOT_TO_UNIT_01.HEARTBEAT := FALSE;
   END_IF;
   "DB7300_INTERLOCK_GENERAL".AUX_SIGNALS_INTERFACE.UNIT_01.LIFE_BIT_FAULT := #_w1 AND (((#COUNTS_FOR_ERROR_UNIT_01 >= 4) AND NOT "DB2031_CYCLES_GENERAL".MANUAL_LOAD_CYCLE.CYCLE_SELECTED) OR ("DB7300_INTERLOCK_GENERAL".AUX_SIGNALS_INTERFACE.UNIT_01.LIFE_BIT_FAULT AND NOT "DB2120_MPP_ITC_IPC".RESET_FAULTS)) AND "DB2120_MPP_ITC_IPC".MACHINE_ON_DELAYED AND "M_DUMMY_OFF";
END_REGION

REGION Network 42: ROBOT FAULT ALARM
   RUNG wire#powerrail
      Contact( "DB7300_INTERLOCK_GENERAL".GENERAL_MACHINE.FROM_ROBOT_TO_UNIT_01.ROBOT_FAULT )
      I_Contact( "DB7300_INTERLOCK_GENERAL".GENERAL_MACHINE.FROM_ROBOT_TO_UNIT_01.OUT_OF_COLLISION_MACHINE )
      wire#w1
      Contact( "DB2120_MPP_ITC_IPC".MACHINE_ON_DELAYED )
      wire#w2
      Coil( "DB7300_INTERLOCK_GENERAL".AUX_SIGNALS_INTERFACE.UNIT_01.ROBOT_FAULT )
   END_RUNG
   RUNG wire#powerrail
      Contact( "DB7300_INTERLOCK_GENERAL".AUX_SIGNALS_INTERFACE.UNIT_01.ROBOT_FAULT )
      I_Contact( "DB2120_MPP_ITC_IPC".RESET_FAULTS )
   END_RUNG wire#w1
   RUNG wire#w2
      Coil( "DB426_ALARMS_WARNINGS".GENERAL."704402" )
   END_RUNG
   // the same network as SCL:
   "DB7300_INTERLOCK_GENERAL".AUX_SIGNALS_INTERFACE.UNIT_01.ROBOT_FAULT := (("DB7300_INTERLOCK_GENERAL".GENERAL_MACHINE.FROM_ROBOT_TO_UNIT_01.ROBOT_FAULT AND NOT "DB7300_INTERLOCK_GENERAL".GENERAL_MACHINE.FROM_ROBOT_TO_UNIT_01.OUT_OF_COLLISION_MACHINE) OR ("DB7300_INTERLOCK_GENERAL".AUX_SIGNALS_INTERFACE.UNIT_01.ROBOT_FAULT AND NOT "DB2120_MPP_ITC_IPC".RESET_FAULTS)) AND "DB2120_MPP_ITC_IPC".MACHINE_ON_DELAYED;
   "DB426_ALARMS_WARNINGS".GENERAL."704402" := "DB7300_INTERLOCK_GENERAL".AUX_SIGNALS_INTERFACE.UNIT_01.ROBOT_FAULT;
END_REGION

REGION Network 44: >>>>>>>>>>>>>>>> INTERLOCKS ROBOT TO MACHINE UNIT 02 <<<<<<<<<<<<<<<<
END_REGION

REGION Network 45: HEARTBEAT
   RUNG wire#powerrail
      Contact( "DB7330_ETXETAR_ROBOT_CELL_INTERLOCK".INTERLOCKS_UNIT_02.ROBOT_TO_MACHINE.RBT_HEARTBEAT )
      Coil( "DB7300_INTERLOCK_GENERAL".GENERAL_MACHINE.FROM_ROBOT_TO_UNIT_02.HEARTBEAT )
   END_RUNG
   // the same network as SCL:
   "DB7300_INTERLOCK_GENERAL".GENERAL_MACHINE.FROM_ROBOT_TO_UNIT_02.HEARTBEAT := "DB7330_ETXETAR_ROBOT_CELL_INTERLOCK".INTERLOCKS_UNIT_02.ROBOT_TO_MACHINE.RBT_HEARTBEAT;
END_REGION

REGION Network 46: EMERGENCY STOP OK
   RUNG wire#powerrail
      Contact( "DB7330_ETXETAR_ROBOT_CELL_INTERLOCK".INTERLOCKS_UNIT_02.ROBOT_TO_MACHINE.RBT_E_STOP_OK )
      Contact( "DB1018_SAFETY_TAGS".CELL_E_STOP_OK )
      wire#w1
      Coil( "DB7300_INTERLOCK_GENERAL".GENERAL_MACHINE.FROM_ROBOT_TO_UNIT_02.EMERG_STOP_OK )
   END_RUNG
   RUNG wire#w1
      Not()
      Coil( "DB7300_INTERLOCK_GENERAL".AUX_SIGNALS_INTERFACE.UNIT_02.EMERGENCY_STOP_ACTIVE )
   END_RUNG
   // the same network as SCL:
   "DB7300_INTERLOCK_GENERAL".GENERAL_MACHINE.FROM_ROBOT_TO_UNIT_02.EMERG_STOP_OK := "DB7330_ETXETAR_ROBOT_CELL_INTERLOCK".INTERLOCKS_UNIT_02.ROBOT_TO_MACHINE.RBT_E_STOP_OK AND "DB1018_SAFETY_TAGS".CELL_E_STOP_OK;
   "DB7300_INTERLOCK_GENERAL".AUX_SIGNALS_INTERFACE.UNIT_02.EMERGENCY_STOP_ACTIVE := NOT "DB7300_INTERLOCK_GENERAL".GENERAL_MACHINE.FROM_ROBOT_TO_UNIT_02.EMERG_STOP_OK;
END_REGION

REGION Network 47: ROBOT FAULT
   RUNG wire#powerrail
      Contact( "DB7330_ETXETAR_ROBOT_CELL_INTERLOCK".INTERLOCKS_UNIT_02.ROBOT_TO_MACHINE.RBT_FAULT )
      Coil( "DB7300_INTERLOCK_GENERAL".GENERAL_MACHINE.FROM_ROBOT_TO_UNIT_02.ROBOT_FAULT )
   END_RUNG
   // the same network as SCL:
   "DB7300_INTERLOCK_GENERAL".GENERAL_MACHINE.FROM_ROBOT_TO_UNIT_02.ROBOT_FAULT := "DB7330_ETXETAR_ROBOT_CELL_INTERLOCK".INTERLOCKS_UNIT_02.ROBOT_TO_MACHINE.RBT_FAULT;
END_REGION

REGION Network 48: GATES CLOSED AND LOCKED
   RUNG wire#powerrail
      Contact( "DB7330_ETXETAR_ROBOT_CELL_INTERLOCK".INTERLOCKS_UNIT_02.ROBOT_TO_MACHINE.RBT_SAFETY_DOOR_CLSD_LCKD )
      wire#w1
      Coil( "DB7300_INTERLOCK_GENERAL".GENERAL_MACHINE.FROM_ROBOT_TO_UNIT_02.SAFETY_DOOR_CLSD_LOCKD )
   END_RUNG
   RUNG wire#powerrail
      Contact( "M_DUMMY_ON" )
   END_RUNG wire#w1
   // the same network as SCL:
   "DB7300_INTERLOCK_GENERAL".GENERAL_MACHINE.FROM_ROBOT_TO_UNIT_02.SAFETY_DOOR_CLSD_LOCKD := "DB7330_ETXETAR_ROBOT_CELL_INTERLOCK".INTERLOCKS_UNIT_02.ROBOT_TO_MACHINE.RBT_SAFETY_DOOR_CLSD_LCKD OR "M_DUMMY_ON";
END_REGION

REGION Network 49: ROBOT CELL EMPTY
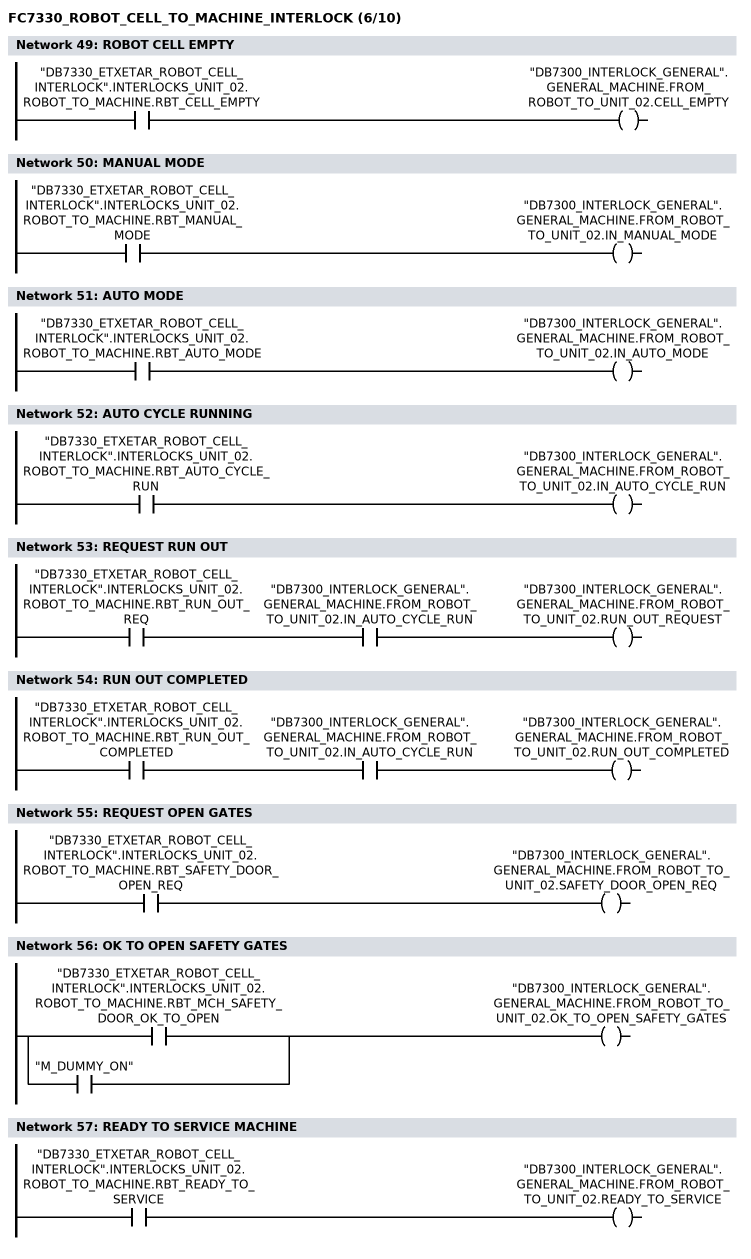
   RUNG wire#powerrail
      Contact( "DB7330_ETXETAR_ROBOT_CELL_INTERLOCK".INTERLOCKS_UNIT_02.ROBOT_TO_MACHINE.RBT_CELL_EMPTY )
      Coil( "DB7300_INTERLOCK_GENERAL".GENERAL_MACHINE.FROM_ROBOT_TO_UNIT_02.CELL_EMPTY )
   END_RUNG
   // the same network as SCL:
   "DB7300_INTERLOCK_GENERAL".GENERAL_MACHINE.FROM_ROBOT_TO_UNIT_02.CELL_EMPTY := "DB7330_ETXETAR_ROBOT_CELL_INTERLOCK".INTERLOCKS_UNIT_02.ROBOT_TO_MACHINE.RBT_CELL_EMPTY;
END_REGION

REGION Network 50: MANUAL MODE
   RUNG wire#powerrail
      Contact( "DB7330_ETXETAR_ROBOT_CELL_INTERLOCK".INTERLOCKS_UNIT_02.ROBOT_TO_MACHINE.RBT_MANUAL_MODE )
      Coil( "DB7300_INTERLOCK_GENERAL".GENERAL_MACHINE.FROM_ROBOT_TO_UNIT_02.IN_MANUAL_MODE )
   END_RUNG
   // the same network as SCL:
   "DB7300_INTERLOCK_GENERAL".GENERAL_MACHINE.FROM_ROBOT_TO_UNIT_02.IN_MANUAL_MODE := "DB7330_ETXETAR_ROBOT_CELL_INTERLOCK".INTERLOCKS_UNIT_02.ROBOT_TO_MACHINE.RBT_MANUAL_MODE;
END_REGION

REGION Network 51: AUTO MODE
   RUNG wire#powerrail
      Contact( "DB7330_ETXETAR_ROBOT_CELL_INTERLOCK".INTERLOCKS_UNIT_02.ROBOT_TO_MACHINE.RBT_AUTO_MODE )
      Coil( "DB7300_INTERLOCK_GENERAL".GENERAL_MACHINE.FROM_ROBOT_TO_UNIT_02.IN_AUTO_MODE )
   END_RUNG
   // the same network as SCL:
   "DB7300_INTERLOCK_GENERAL".GENERAL_MACHINE.FROM_ROBOT_TO_UNIT_02.IN_AUTO_MODE := "DB7330_ETXETAR_ROBOT_CELL_INTERLOCK".INTERLOCKS_UNIT_02.ROBOT_TO_MACHINE.RBT_AUTO_MODE;
END_REGION

REGION Network 52: AUTO CYCLE RUNNING
   RUNG wire#powerrail
      Contact( "DB7330_ETXETAR_ROBOT_CELL_INTERLOCK".INTERLOCKS_UNIT_02.ROBOT_TO_MACHINE.RBT_AUTO_CYCLE_RUN )
      Coil( "DB7300_INTERLOCK_GENERAL".GENERAL_MACHINE.FROM_ROBOT_TO_UNIT_02.IN_AUTO_CYCLE_RUN )
   END_RUNG
   // the same network as SCL:
   "DB7300_INTERLOCK_GENERAL".GENERAL_MACHINE.FROM_ROBOT_TO_UNIT_02.IN_AUTO_CYCLE_RUN := "DB7330_ETXETAR_ROBOT_CELL_INTERLOCK".INTERLOCKS_UNIT_02.ROBOT_TO_MACHINE.RBT_AUTO_CYCLE_RUN;
END_REGION

REGION Network 53: REQUEST RUN OUT
   RUNG wire#powerrail
      Contact( "DB7330_ETXETAR_ROBOT_CELL_INTERLOCK".INTERLOCKS_UNIT_02.ROBOT_TO_MACHINE.RBT_RUN_OUT_REQ )
      Contact( "DB7300_INTERLOCK_GENERAL".GENERAL_MACHINE.FROM_ROBOT_TO_UNIT_02.IN_AUTO_CYCLE_RUN )
      Coil( "DB7300_INTERLOCK_GENERAL".GENERAL_MACHINE.FROM_ROBOT_TO_UNIT_02.RUN_OUT_REQUEST )
   END_RUNG
   // the same network as SCL:
   "DB7300_INTERLOCK_GENERAL".GENERAL_MACHINE.FROM_ROBOT_TO_UNIT_02.RUN_OUT_REQUEST := "DB7330_ETXETAR_ROBOT_CELL_INTERLOCK".INTERLOCKS_UNIT_02.ROBOT_TO_MACHINE.RBT_RUN_OUT_REQ AND "DB7300_INTERLOCK_GENERAL".GENERAL_MACHINE.FROM_ROBOT_TO_UNIT_02.IN_AUTO_CYCLE_RUN;
END_REGION

REGION Network 54: RUN OUT COMPLETED
   RUNG wire#powerrail
      Contact( "DB7330_ETXETAR_ROBOT_CELL_INTERLOCK".INTERLOCKS_UNIT_02.ROBOT_TO_MACHINE.RBT_RUN_OUT_COMPLETED )
      Contact( "DB7300_INTERLOCK_GENERAL".GENERAL_MACHINE.FROM_ROBOT_TO_UNIT_02.IN_AUTO_CYCLE_RUN )
      Coil( "DB7300_INTERLOCK_GENERAL".GENERAL_MACHINE.FROM_ROBOT_TO_UNIT_02.RUN_OUT_COMPLETED )
   END_RUNG
   // the same network as SCL:
   "DB7300_INTERLOCK_GENERAL".GENERAL_MACHINE.FROM_ROBOT_TO_UNIT_02.RUN_OUT_COMPLETED := "DB7330_ETXETAR_ROBOT_CELL_INTERLOCK".INTERLOCKS_UNIT_02.ROBOT_TO_MACHINE.RBT_RUN_OUT_COMPLETED AND "DB7300_INTERLOCK_GENERAL".GENERAL_MACHINE.FROM_ROBOT_TO_UNIT_02.IN_AUTO_CYCLE_RUN;
END_REGION

REGION Network 55: REQUEST OPEN GATES
   RUNG wire#powerrail
      Contact( "DB7330_ETXETAR_ROBOT_CELL_INTERLOCK".INTERLOCKS_UNIT_02.ROBOT_TO_MACHINE.RBT_SAFETY_DOOR_OPEN_REQ )
      Coil( "DB7300_INTERLOCK_GENERAL".GENERAL_MACHINE.FROM_ROBOT_TO_UNIT_02.SAFETY_DOOR_OPEN_REQ )
   END_RUNG
   // the same network as SCL:
   "DB7300_INTERLOCK_GENERAL".GENERAL_MACHINE.FROM_ROBOT_TO_UNIT_02.SAFETY_DOOR_OPEN_REQ := "DB7330_ETXETAR_ROBOT_CELL_INTERLOCK".INTERLOCKS_UNIT_02.ROBOT_TO_MACHINE.RBT_SAFETY_DOOR_OPEN_REQ;
END_REGION

REGION Network 56: OK TO OPEN SAFETY GATES
   RUNG wire#powerrail
      Contact( "DB7330_ETXETAR_ROBOT_CELL_INTERLOCK".INTERLOCKS_UNIT_02.ROBOT_TO_MACHINE.RBT_MCH_SAFETY_DOOR_OK_TO_OPEN )
      wire#w1
      Coil( "DB7300_INTERLOCK_GENERAL".GENERAL_MACHINE.FROM_ROBOT_TO_UNIT_02.OK_TO_OPEN_SAFETY_GATES )
   END_RUNG
   RUNG wire#powerrail
      Contact( "M_DUMMY_ON" )
   END_RUNG wire#w1
   // the same network as SCL:
   "DB7300_INTERLOCK_GENERAL".GENERAL_MACHINE.FROM_ROBOT_TO_UNIT_02.OK_TO_OPEN_SAFETY_GATES := "DB7330_ETXETAR_ROBOT_CELL_INTERLOCK".INTERLOCKS_UNIT_02.ROBOT_TO_MACHINE.RBT_MCH_SAFETY_DOOR_OK_TO_OPEN OR "M_DUMMY_ON";
END_REGION

REGION Network 57: READY TO SERVICE MACHINE
   RUNG wire#powerrail
      Contact( "DB7330_ETXETAR_ROBOT_CELL_INTERLOCK".INTERLOCKS_UNIT_02.ROBOT_TO_MACHINE.RBT_READY_TO_SERVICE )
      Coil( "DB7300_INTERLOCK_GENERAL".GENERAL_MACHINE.FROM_ROBOT_TO_UNIT_02.READY_TO_SERVICE )
   END_RUNG
   // the same network as SCL:
   "DB7300_INTERLOCK_GENERAL".GENERAL_MACHINE.FROM_ROBOT_TO_UNIT_02.READY_TO_SERVICE := "DB7330_ETXETAR_ROBOT_CELL_INTERLOCK".INTERLOCKS_UNIT_02.ROBOT_TO_MACHINE.RBT_READY_TO_SERVICE;
END_REGION

REGION Network 58: OUT OF COLLISION MACHINE
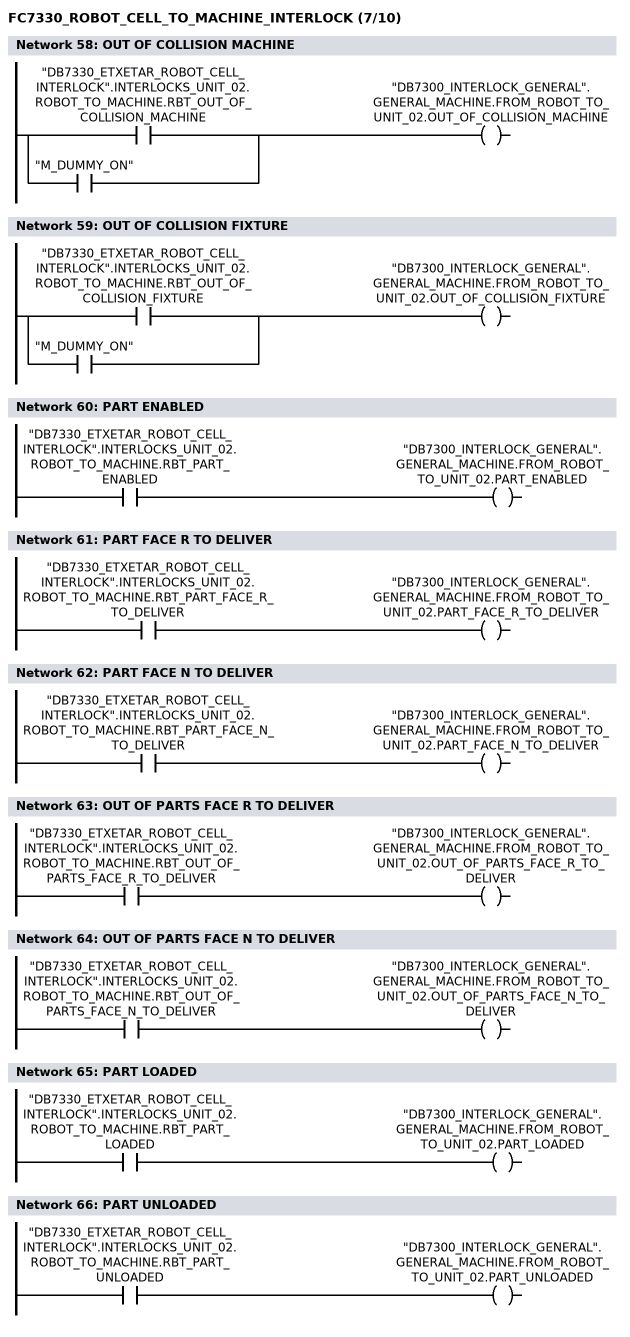
   RUNG wire#powerrail
      Contact( "DB7330_ETXETAR_ROBOT_CELL_INTERLOCK".INTERLOCKS_UNIT_02.ROBOT_TO_MACHINE.RBT_OUT_OF_COLLISION_MACHINE )
      wire#w1
      Coil( "DB7300_INTERLOCK_GENERAL".GENERAL_MACHINE.FROM_ROBOT_TO_UNIT_02.OUT_OF_COLLISION_MACHINE )
   END_RUNG
   RUNG wire#powerrail
      Contact( "M_DUMMY_ON" )
   END_RUNG wire#w1
   // the same network as SCL:
   "DB7300_INTERLOCK_GENERAL".GENERAL_MACHINE.FROM_ROBOT_TO_UNIT_02.OUT_OF_COLLISION_MACHINE := "DB7330_ETXETAR_ROBOT_CELL_INTERLOCK".INTERLOCKS_UNIT_02.ROBOT_TO_MACHINE.RBT_OUT_OF_COLLISION_MACHINE OR "M_DUMMY_ON";
END_REGION

REGION Network 59: OUT OF COLLISION FIXTURE
   RUNG wire#powerrail
      Contact( "DB7330_ETXETAR_ROBOT_CELL_INTERLOCK".INTERLOCKS_UNIT_02.ROBOT_TO_MACHINE.RBT_OUT_OF_COLLISION_FIXTURE )
      wire#w1
      Coil( "DB7300_INTERLOCK_GENERAL".GENERAL_MACHINE.FROM_ROBOT_TO_UNIT_02.OUT_OF_COLLISION_FIXTURE )
   END_RUNG
   RUNG wire#powerrail
      Contact( "M_DUMMY_ON" )
   END_RUNG wire#w1
   // the same network as SCL:
   "DB7300_INTERLOCK_GENERAL".GENERAL_MACHINE.FROM_ROBOT_TO_UNIT_02.OUT_OF_COLLISION_FIXTURE := "DB7330_ETXETAR_ROBOT_CELL_INTERLOCK".INTERLOCKS_UNIT_02.ROBOT_TO_MACHINE.RBT_OUT_OF_COLLISION_FIXTURE OR "M_DUMMY_ON";
END_REGION

REGION Network 60: PART ENABLED
   RUNG wire#powerrail
      Contact( "DB7330_ETXETAR_ROBOT_CELL_INTERLOCK".INTERLOCKS_UNIT_02.ROBOT_TO_MACHINE.RBT_PART_ENABLED )
      Coil( "DB7300_INTERLOCK_GENERAL".GENERAL_MACHINE.FROM_ROBOT_TO_UNIT_02.PART_ENABLED )
   END_RUNG
   // the same network as SCL:
   "DB7300_INTERLOCK_GENERAL".GENERAL_MACHINE.FROM_ROBOT_TO_UNIT_02.PART_ENABLED := "DB7330_ETXETAR_ROBOT_CELL_INTERLOCK".INTERLOCKS_UNIT_02.ROBOT_TO_MACHINE.RBT_PART_ENABLED;
END_REGION

REGION Network 61: PART FACE R TO DELIVER
   RUNG wire#powerrail
      Contact( "DB7330_ETXETAR_ROBOT_CELL_INTERLOCK".INTERLOCKS_UNIT_02.ROBOT_TO_MACHINE.RBT_PART_FACE_R_TO_DELIVER )
      Coil( "DB7300_INTERLOCK_GENERAL".GENERAL_MACHINE.FROM_ROBOT_TO_UNIT_02.PART_FACE_R_TO_DELIVER )
   END_RUNG
   // the same network as SCL:
   "DB7300_INTERLOCK_GENERAL".GENERAL_MACHINE.FROM_ROBOT_TO_UNIT_02.PART_FACE_R_TO_DELIVER := "DB7330_ETXETAR_ROBOT_CELL_INTERLOCK".INTERLOCKS_UNIT_02.ROBOT_TO_MACHINE.RBT_PART_FACE_R_TO_DELIVER;
END_REGION

REGION Network 62: PART FACE N TO DELIVER
   RUNG wire#powerrail
      Contact( "DB7330_ETXETAR_ROBOT_CELL_INTERLOCK".INTERLOCKS_UNIT_02.ROBOT_TO_MACHINE.RBT_PART_FACE_N_TO_DELIVER )
      Coil( "DB7300_INTERLOCK_GENERAL".GENERAL_MACHINE.FROM_ROBOT_TO_UNIT_02.PART_FACE_N_TO_DELIVER )
   END_RUNG
   // the same network as SCL:
   "DB7300_INTERLOCK_GENERAL".GENERAL_MACHINE.FROM_ROBOT_TO_UNIT_02.PART_FACE_N_TO_DELIVER := "DB7330_ETXETAR_ROBOT_CELL_INTERLOCK".INTERLOCKS_UNIT_02.ROBOT_TO_MACHINE.RBT_PART_FACE_N_TO_DELIVER;
END_REGION

REGION Network 63: OUT OF PARTS FACE R TO DELIVER
   RUNG wire#powerrail
      Contact( "DB7330_ETXETAR_ROBOT_CELL_INTERLOCK".INTERLOCKS_UNIT_02.ROBOT_TO_MACHINE.RBT_OUT_OF_PARTS_FACE_R_TO_DELIVER )
      Coil( "DB7300_INTERLOCK_GENERAL".GENERAL_MACHINE.FROM_ROBOT_TO_UNIT_02.OUT_OF_PARTS_FACE_R_TO_DELIVER )
   END_RUNG
   // the same network as SCL:
   "DB7300_INTERLOCK_GENERAL".GENERAL_MACHINE.FROM_ROBOT_TO_UNIT_02.OUT_OF_PARTS_FACE_R_TO_DELIVER := "DB7330_ETXETAR_ROBOT_CELL_INTERLOCK".INTERLOCKS_UNIT_02.ROBOT_TO_MACHINE.RBT_OUT_OF_PARTS_FACE_R_TO_DELIVER;
END_REGION

REGION Network 64: OUT OF PARTS FACE N TO DELIVER
   RUNG wire#powerrail
      Contact( "DB7330_ETXETAR_ROBOT_CELL_INTERLOCK".INTERLOCKS_UNIT_02.ROBOT_TO_MACHINE.RBT_OUT_OF_PARTS_FACE_N_TO_DELIVER )
      Coil( "DB7300_INTERLOCK_GENERAL".GENERAL_MACHINE.FROM_ROBOT_TO_UNIT_02.OUT_OF_PARTS_FACE_N_TO_DELIVER )
   END_RUNG
   // the same network as SCL:
   "DB7300_INTERLOCK_GENERAL".GENERAL_MACHINE.FROM_ROBOT_TO_UNIT_02.OUT_OF_PARTS_FACE_N_TO_DELIVER := "DB7330_ETXETAR_ROBOT_CELL_INTERLOCK".INTERLOCKS_UNIT_02.ROBOT_TO_MACHINE.RBT_OUT_OF_PARTS_FACE_N_TO_DELIVER;
END_REGION

REGION Network 65: PART LOADED
   RUNG wire#powerrail
      Contact( "DB7330_ETXETAR_ROBOT_CELL_INTERLOCK".INTERLOCKS_UNIT_02.ROBOT_TO_MACHINE.RBT_PART_LOADED )
      Coil( "DB7300_INTERLOCK_GENERAL".GENERAL_MACHINE.FROM_ROBOT_TO_UNIT_02.PART_LOADED )
   END_RUNG
   // the same network as SCL:
   "DB7300_INTERLOCK_GENERAL".GENERAL_MACHINE.FROM_ROBOT_TO_UNIT_02.PART_LOADED := "DB7330_ETXETAR_ROBOT_CELL_INTERLOCK".INTERLOCKS_UNIT_02.ROBOT_TO_MACHINE.RBT_PART_LOADED;
END_REGION

REGION Network 66: PART UNLOADED
   RUNG wire#powerrail
      Contact( "DB7330_ETXETAR_ROBOT_CELL_INTERLOCK".INTERLOCKS_UNIT_02.ROBOT_TO_MACHINE.RBT_PART_UNLOADED )
      Coil( "DB7300_INTERLOCK_GENERAL".GENERAL_MACHINE.FROM_ROBOT_TO_UNIT_02.PART_UNLOADED )
   END_RUNG
   // the same network as SCL:
   "DB7300_INTERLOCK_GENERAL".GENERAL_MACHINE.FROM_ROBOT_TO_UNIT_02.PART_UNLOADED := "DB7330_ETXETAR_ROBOT_CELL_INTERLOCK".INTERLOCKS_UNIT_02.ROBOT_TO_MACHINE.RBT_PART_UNLOADED;
END_REGION

REGION Network 67: FIXTURE SKIP REQUEST
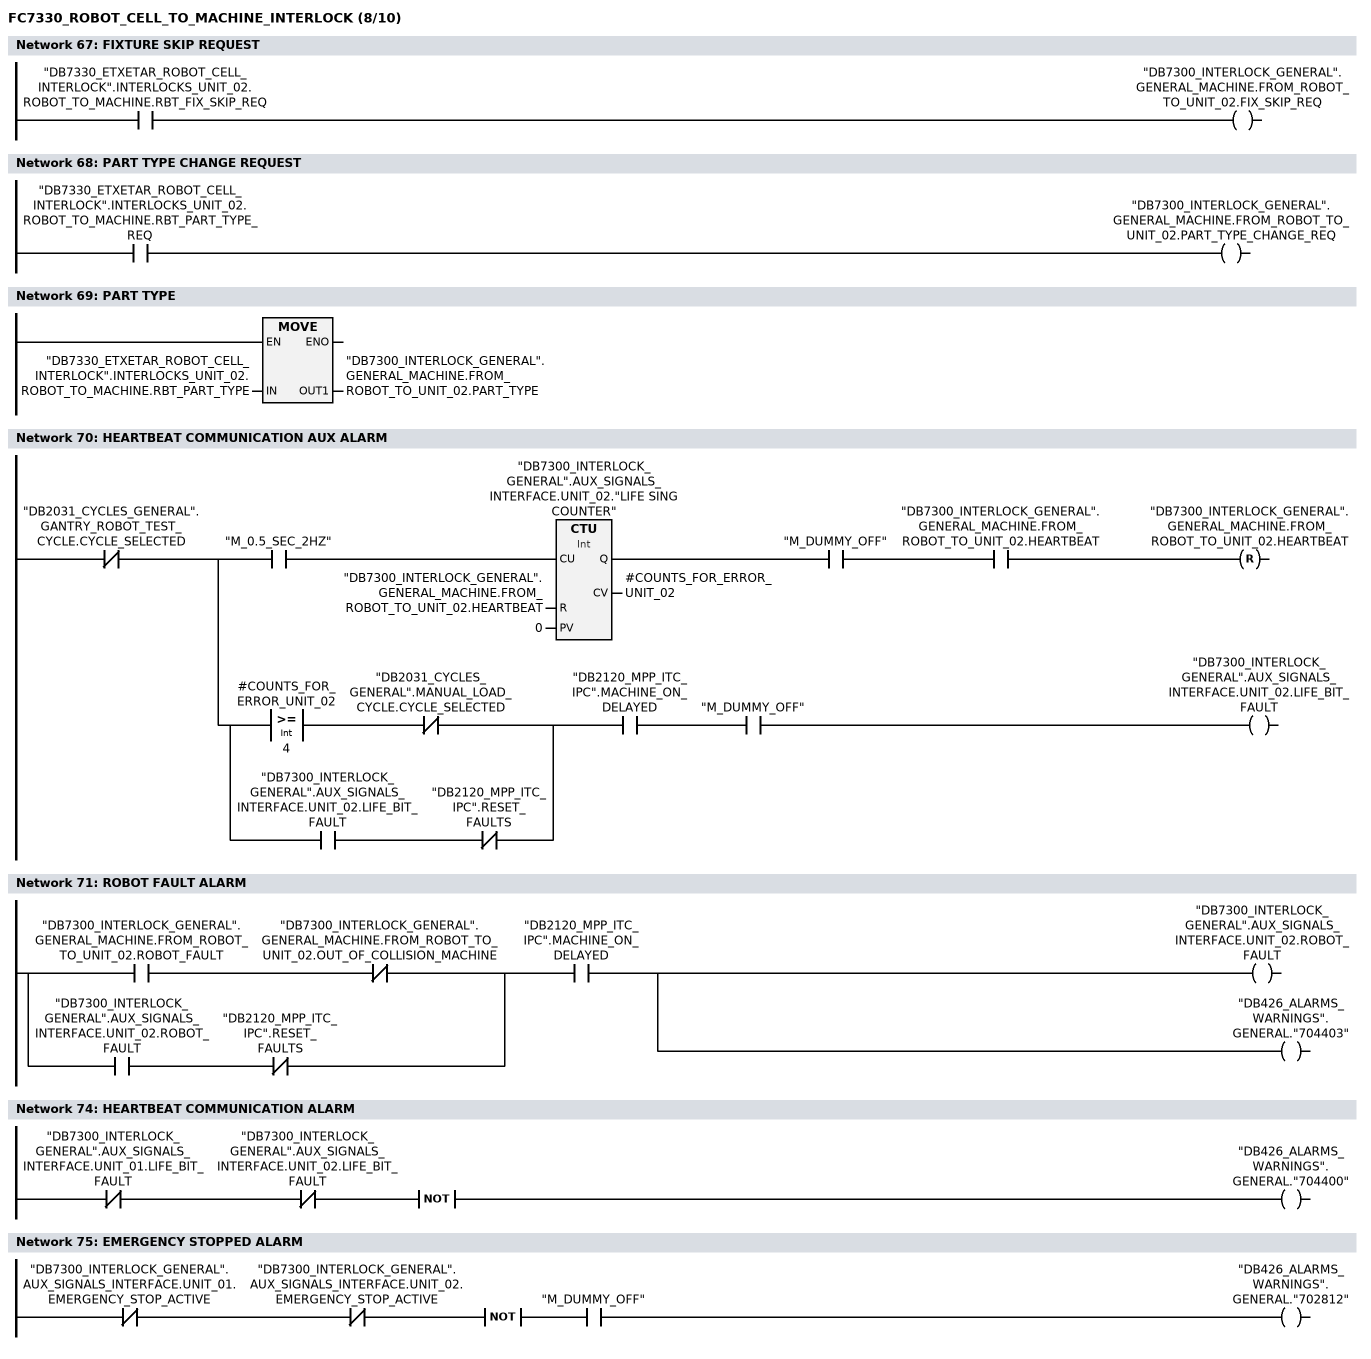
   RUNG wire#powerrail
      Contact( "DB7330_ETXETAR_ROBOT_CELL_INTERLOCK".INTERLOCKS_UNIT_02.ROBOT_TO_MACHINE.RBT_FIX_SKIP_REQ )
      Coil( "DB7300_INTERLOCK_GENERAL".GENERAL_MACHINE.FROM_ROBOT_TO_UNIT_02.FIX_SKIP_REQ )
   END_RUNG
   // the same network as SCL:
   "DB7300_INTERLOCK_GENERAL".GENERAL_MACHINE.FROM_ROBOT_TO_UNIT_02.FIX_SKIP_REQ := "DB7330_ETXETAR_ROBOT_CELL_INTERLOCK".INTERLOCKS_UNIT_02.ROBOT_TO_MACHINE.RBT_FIX_SKIP_REQ;
END_REGION

REGION Network 68: PART TYPE CHANGE REQUEST
   RUNG wire#powerrail
      Contact( "DB7330_ETXETAR_ROBOT_CELL_INTERLOCK".INTERLOCKS_UNIT_02.ROBOT_TO_MACHINE.RBT_PART_TYPE_REQ )
      Coil( "DB7300_INTERLOCK_GENERAL".GENERAL_MACHINE.FROM_ROBOT_TO_UNIT_02.PART_TYPE_CHANGE_REQ )
   END_RUNG
   // the same network as SCL:
   "DB7300_INTERLOCK_GENERAL".GENERAL_MACHINE.FROM_ROBOT_TO_UNIT_02.PART_TYPE_CHANGE_REQ := "DB7330_ETXETAR_ROBOT_CELL_INTERLOCK".INTERLOCKS_UNIT_02.ROBOT_TO_MACHINE.RBT_PART_TYPE_REQ;
END_REGION

REGION Network 69: PART TYPE
   RUNG wire#powerrail
      { S7_GenerateENO := "TRUE" } Move(in := "DB7330_ETXETAR_ROBOT_CELL_INTERLOCK".INTERLOCKS_UNIT_02.ROBOT_TO_MACHINE.RBT_PART_TYPE, out1 => "DB7300_INTERLOCK_GENERAL".GENERAL_MACHINE.FROM_ROBOT_TO_UNIT_02.PART_TYPE)
   END_RUNG
   // the same network as SCL:
   "DB7300_INTERLOCK_GENERAL".GENERAL_MACHINE.FROM_ROBOT_TO_UNIT_02.PART_TYPE := "DB7330_ETXETAR_ROBOT_CELL_INTERLOCK".INTERLOCKS_UNIT_02.ROBOT_TO_MACHINE.RBT_PART_TYPE;
END_REGION

REGION Network 70: HEARTBEAT COMMUNICATION AUX ALARM
   RUNG wire#powerrail
      I_Contact( "DB2031_CYCLES_GENERAL".GANTRY_ROBOT_TEST_CYCLE.CYCLE_SELECTED )
      wire#w1
      Contact( "M_0.5_SEC_2HZ" )
      { S7_Templates := "value_type := Int" } "DB7300_INTERLOCK_GENERAL".AUX_SIGNALS_INTERFACE.UNIT_02."LIFE SING COUNTER".CTU(r := "DB7300_INTERLOCK_GENERAL".GENERAL_MACHINE.FROM_ROBOT_TO_UNIT_02.HEARTBEAT, pv := 0, cv => #COUNTS_FOR_ERROR_UNIT_02)
      Contact( "M_DUMMY_OFF" )
      Contact( "DB7300_INTERLOCK_GENERAL".GENERAL_MACHINE.FROM_ROBOT_TO_UNIT_02.HEARTBEAT )
      R_Coil( "DB7300_INTERLOCK_GENERAL".GENERAL_MACHINE.FROM_ROBOT_TO_UNIT_02.HEARTBEAT )
   END_RUNG
   RUNG wire#w1
      { S7_Templates := "SrcType := Int" } GE_Contact(in1 := #COUNTS_FOR_ERROR_UNIT_02, in2 := 4)
      I_Contact( "DB2031_CYCLES_GENERAL".MANUAL_LOAD_CYCLE.CYCLE_SELECTED )
      wire#w2
      Contact( "DB2120_MPP_ITC_IPC".MACHINE_ON_DELAYED )
      Contact( "M_DUMMY_OFF" )
      Coil( "DB7300_INTERLOCK_GENERAL".AUX_SIGNALS_INTERFACE.UNIT_02.LIFE_BIT_FAULT )
   END_RUNG
   RUNG wire#w1
      Contact( "DB7300_INTERLOCK_GENERAL".AUX_SIGNALS_INTERFACE.UNIT_02.LIFE_BIT_FAULT )
      I_Contact( "DB2120_MPP_ITC_IPC".RESET_FAULTS )
   END_RUNG wire#w2
   // the same network as SCL:
   #_w1 := NOT "DB2031_CYCLES_GENERAL".GANTRY_ROBOT_TEST_CYCLE.CYCLE_SELECTED;
   "DB7300_INTERLOCK_GENERAL".AUX_SIGNALS_INTERFACE.UNIT_02."LIFE SING COUNTER".CTU(CU := #_w1 AND "M_0.5_SEC_2HZ",
                           R := "DB7300_INTERLOCK_GENERAL".GENERAL_MACHINE.FROM_ROBOT_TO_UNIT_02.HEARTBEAT,
                           PV := 0,
                           CV => #COUNTS_FOR_ERROR_UNIT_02);
   IF "DB7300_INTERLOCK_GENERAL".AUX_SIGNALS_INTERFACE.UNIT_02."LIFE SING COUNTER".Q AND "M_DUMMY_OFF" AND "DB7300_INTERLOCK_GENERAL".GENERAL_MACHINE.FROM_ROBOT_TO_UNIT_02.HEARTBEAT THEN
       "DB7300_INTERLOCK_GENERAL".GENERAL_MACHINE.FROM_ROBOT_TO_UNIT_02.HEARTBEAT := FALSE;
   END_IF;
   "DB7300_INTERLOCK_GENERAL".AUX_SIGNALS_INTERFACE.UNIT_02.LIFE_BIT_FAULT := #_w1 AND (((#COUNTS_FOR_ERROR_UNIT_02 >= 4) AND NOT "DB2031_CYCLES_GENERAL".MANUAL_LOAD_CYCLE.CYCLE_SELECTED) OR ("DB7300_INTERLOCK_GENERAL".AUX_SIGNALS_INTERFACE.UNIT_02.LIFE_BIT_FAULT AND NOT "DB2120_MPP_ITC_IPC".RESET_FAULTS)) AND "DB2120_MPP_ITC_IPC".MACHINE_ON_DELAYED AND "M_DUMMY_OFF";
END_REGION

REGION Network 71: ROBOT FAULT ALARM
   RUNG wire#powerrail
      Contact( "DB7300_INTERLOCK_GENERAL".GENERAL_MACHINE.FROM_ROBOT_TO_UNIT_02.ROBOT_FAULT )
      I_Contact( "DB7300_INTERLOCK_GENERAL".GENERAL_MACHINE.FROM_ROBOT_TO_UNIT_02.OUT_OF_COLLISION_MACHINE )
      wire#w1
      Contact( "DB2120_MPP_ITC_IPC".MACHINE_ON_DELAYED )
      wire#w2
      Coil( "DB7300_INTERLOCK_GENERAL".AUX_SIGNALS_INTERFACE.UNIT_02.ROBOT_FAULT )
   END_RUNG
   RUNG wire#powerrail
      Contact( "DB7300_INTERLOCK_GENERAL".AUX_SIGNALS_INTERFACE.UNIT_02.ROBOT_FAULT )
      I_Contact( "DB2120_MPP_ITC_IPC".RESET_FAULTS )
   END_RUNG wire#w1
   RUNG wire#w2
      Coil( "DB426_ALARMS_WARNINGS".GENERAL."704403" )
   END_RUNG
   // the same network as SCL:
   "DB7300_INTERLOCK_GENERAL".AUX_SIGNALS_INTERFACE.UNIT_02.ROBOT_FAULT := (("DB7300_INTERLOCK_GENERAL".GENERAL_MACHINE.FROM_ROBOT_TO_UNIT_02.ROBOT_FAULT AND NOT "DB7300_INTERLOCK_GENERAL".GENERAL_MACHINE.FROM_ROBOT_TO_UNIT_02.OUT_OF_COLLISION_MACHINE) OR ("DB7300_INTERLOCK_GENERAL".AUX_SIGNALS_INTERFACE.UNIT_02.ROBOT_FAULT AND NOT "DB2120_MPP_ITC_IPC".RESET_FAULTS)) AND "DB2120_MPP_ITC_IPC".MACHINE_ON_DELAYED;
   "DB426_ALARMS_WARNINGS".GENERAL."704403" := "DB7300_INTERLOCK_GENERAL".AUX_SIGNALS_INTERFACE.UNIT_02.ROBOT_FAULT;
END_REGION

REGION Network 73: >>>>>>>>>>>>>>>> INTERLOCKS ALARMS & WARNINGS <<<<<<<<<<<<<<<<
END_REGION

REGION Network 74: HEARTBEAT COMMUNICATION ALARM
   RUNG wire#powerrail
      I_Contact( "DB7300_INTERLOCK_GENERAL".AUX_SIGNALS_INTERFACE.UNIT_01.LIFE_BIT_FAULT )
      I_Contact( "DB7300_INTERLOCK_GENERAL".AUX_SIGNALS_INTERFACE.UNIT_02.LIFE_BIT_FAULT )
      Not()
      Coil( "DB426_ALARMS_WARNINGS".GENERAL."704400" )
   END_RUNG
   // the same network as SCL:
   "DB426_ALARMS_WARNINGS".GENERAL."704400" := NOT (NOT "DB7300_INTERLOCK_GENERAL".AUX_SIGNALS_INTERFACE.UNIT_01.LIFE_BIT_FAULT AND NOT "DB7300_INTERLOCK_GENERAL".AUX_SIGNALS_INTERFACE.UNIT_02.LIFE_BIT_FAULT);
END_REGION

REGION Network 75: EMERGENCY STOPPED ALARM
   RUNG wire#powerrail
      I_Contact( "DB7300_INTERLOCK_GENERAL".AUX_SIGNALS_INTERFACE.UNIT_01.EMERGENCY_STOP_ACTIVE )
      I_Contact( "DB7300_INTERLOCK_GENERAL".AUX_SIGNALS_INTERFACE.UNIT_02.EMERGENCY_STOP_ACTIVE )
      Not()
      Contact( "M_DUMMY_OFF" )
      Coil( "DB426_ALARMS_WARNINGS".GENERAL."702812" )
   END_RUNG
   // the same network as SCL:
   "DB426_ALARMS_WARNINGS".GENERAL."702812" := NOT (NOT "DB7300_INTERLOCK_GENERAL".AUX_SIGNALS_INTERFACE.UNIT_01.EMERGENCY_STOP_ACTIVE AND NOT "DB7300_INTERLOCK_GENERAL".AUX_SIGNALS_INTERFACE.UNIT_02.EMERGENCY_STOP_ACTIVE) AND "M_DUMMY_OFF";
END_REGION

REGION Network 76: MEASURING STATION FAULT ALARM
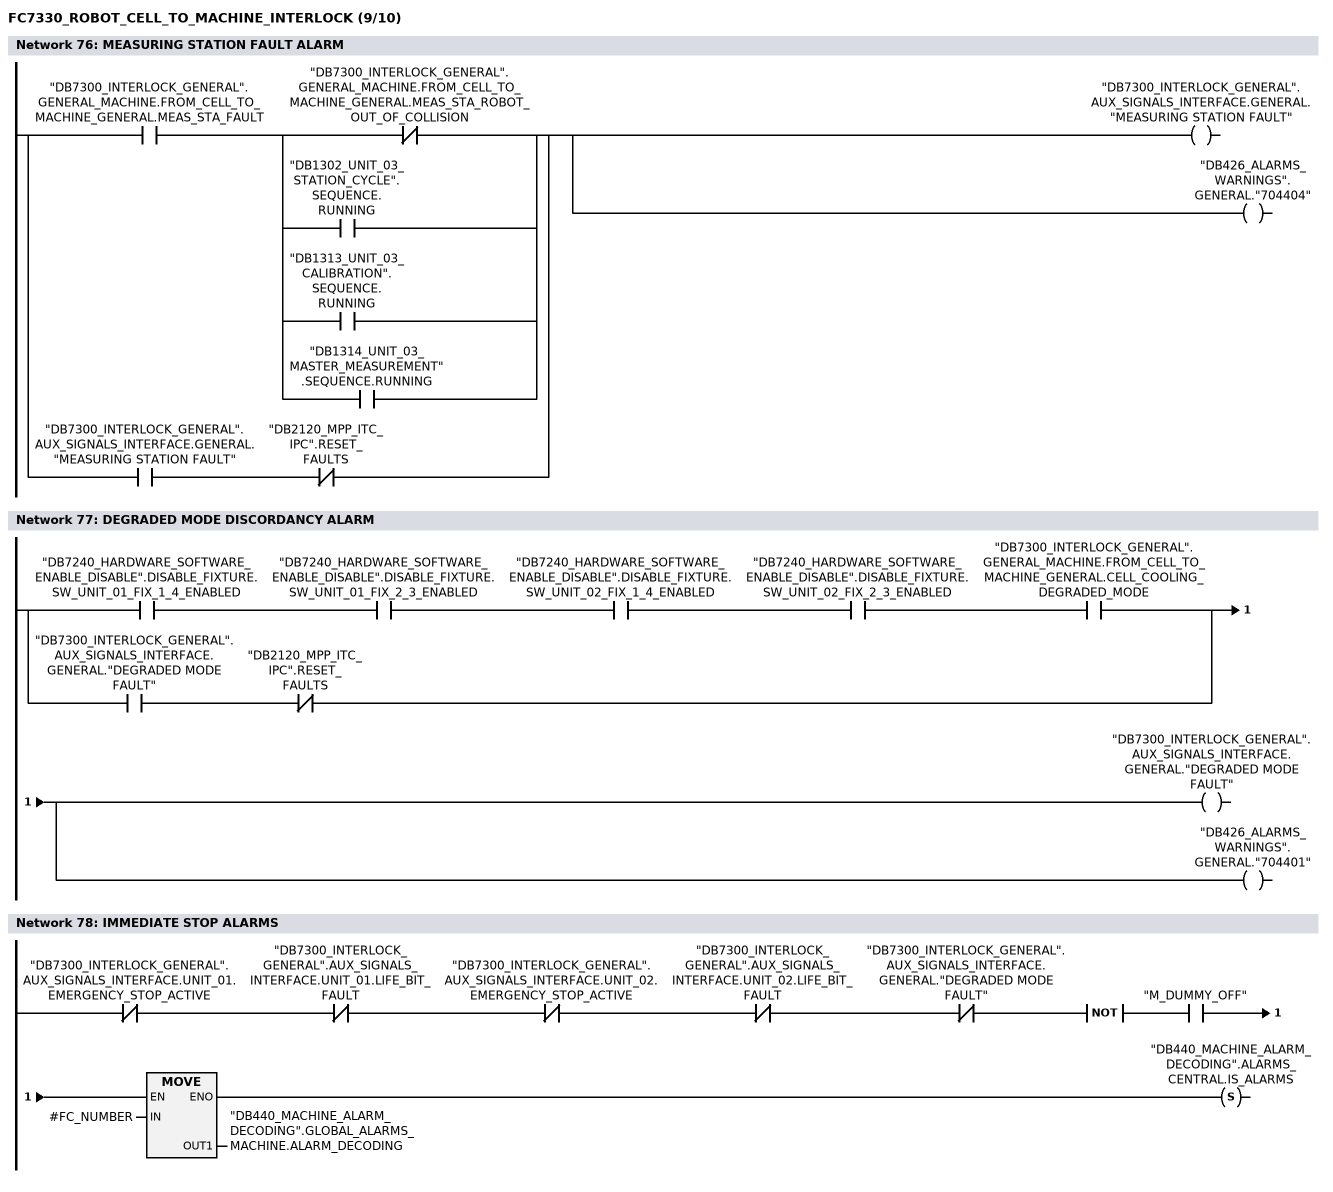
   RUNG wire#powerrail
      Contact( "DB7300_INTERLOCK_GENERAL".GENERAL_MACHINE.FROM_CELL_TO_MACHINE_GENERAL.MEAS_STA_FAULT )
      wire#w1
      I_Contact( "DB7300_INTERLOCK_GENERAL".GENERAL_MACHINE.FROM_CELL_TO_MACHINE_GENERAL.MEAS_STA_ROBOT_OUT_OF_COLLISION )
      wire#w2
      Coil( "DB7300_INTERLOCK_GENERAL".AUX_SIGNALS_INTERFACE.GENERAL."MEASURING STATION FAULT" )
   END_RUNG
   RUNG wire#w1
      Contact( "DB1302_UNIT_03_STATION_CYCLE".SEQUENCE.RUNNING )
   END_RUNG wire#w2
   RUNG wire#w1
      Contact( "DB1313_UNIT_03_CALIBRATION".SEQUENCE.RUNNING )
   END_RUNG wire#w2
   RUNG wire#w1
      Contact( "DB1314_UNIT_03_MASTER_MEASUREMENT".SEQUENCE.RUNNING )
   END_RUNG wire#w2
   RUNG wire#powerrail
      Contact( "DB7300_INTERLOCK_GENERAL".AUX_SIGNALS_INTERFACE.GENERAL."MEASURING STATION FAULT" )
      I_Contact( "DB2120_MPP_ITC_IPC".RESET_FAULTS )
   END_RUNG wire#w2
   RUNG wire#w2
      Coil( "DB426_ALARMS_WARNINGS".GENERAL."704404" )
   END_RUNG
   // the same network as SCL:
   "DB7300_INTERLOCK_GENERAL".AUX_SIGNALS_INTERFACE.GENERAL."MEASURING STATION FAULT" := ("DB7300_INTERLOCK_GENERAL".GENERAL_MACHINE.FROM_CELL_TO_MACHINE_GENERAL.MEAS_STA_FAULT AND (NOT "DB7300_INTERLOCK_GENERAL".GENERAL_MACHINE.FROM_CELL_TO_MACHINE_GENERAL.MEAS_STA_ROBOT_OUT_OF_COLLISION OR "DB1302_UNIT_03_STATION_CYCLE".SEQUENCE.RUNNING OR "DB1313_UNIT_03_CALIBRATION".SEQUENCE.RUNNING OR "DB1314_UNIT_03_MASTER_MEASUREMENT".SEQUENCE.RUNNING)) OR ("DB7300_INTERLOCK_GENERAL".AUX_SIGNALS_INTERFACE.GENERAL."MEASURING STATION FAULT" AND NOT "DB2120_MPP_ITC_IPC".RESET_FAULTS);
   "DB426_ALARMS_WARNINGS".GENERAL."704404" := "DB7300_INTERLOCK_GENERAL".AUX_SIGNALS_INTERFACE.GENERAL."MEASURING STATION FAULT";
END_REGION

REGION Network 77: DEGRADED MODE DISCORDANCY ALARM
   RUNG wire#powerrail
      Contact( "DB7240_HARDWARE_SOFTWARE_ENABLE_DISABLE".DISABLE_FIXTURE.SW_UNIT_01_FIX_1_4_ENABLED )
      Contact( "DB7240_HARDWARE_SOFTWARE_ENABLE_DISABLE".DISABLE_FIXTURE.SW_UNIT_01_FIX_2_3_ENABLED )
      Contact( "DB7240_HARDWARE_SOFTWARE_ENABLE_DISABLE".DISABLE_FIXTURE.SW_UNIT_02_FIX_1_4_ENABLED )
      Contact( "DB7240_HARDWARE_SOFTWARE_ENABLE_DISABLE".DISABLE_FIXTURE.SW_UNIT_02_FIX_2_3_ENABLED )
      Contact( "DB7300_INTERLOCK_GENERAL".GENERAL_MACHINE.FROM_CELL_TO_MACHINE_GENERAL.CELL_COOLING_DEGRADED_MODE )
      wire#w1
      Coil( "DB7300_INTERLOCK_GENERAL".AUX_SIGNALS_INTERFACE.GENERAL."DEGRADED MODE FAULT" )
   END_RUNG
   RUNG wire#powerrail
      Contact( "DB7300_INTERLOCK_GENERAL".AUX_SIGNALS_INTERFACE.GENERAL."DEGRADED MODE FAULT" )
      I_Contact( "DB2120_MPP_ITC_IPC".RESET_FAULTS )
   END_RUNG wire#w1
   RUNG wire#w1
      Coil( "DB426_ALARMS_WARNINGS".GENERAL."704401" )
   END_RUNG
   // the same network as SCL:
   "DB7300_INTERLOCK_GENERAL".AUX_SIGNALS_INTERFACE.GENERAL."DEGRADED MODE FAULT" := ("DB7240_HARDWARE_SOFTWARE_ENABLE_DISABLE".DISABLE_FIXTURE.SW_UNIT_01_FIX_1_4_ENABLED AND "DB7240_HARDWARE_SOFTWARE_ENABLE_DISABLE".DISABLE_FIXTURE.SW_UNIT_01_FIX_2_3_ENABLED AND "DB7240_HARDWARE_SOFTWARE_ENABLE_DISABLE".DISABLE_FIXTURE.SW_UNIT_02_FIX_1_4_ENABLED AND "DB7240_HARDWARE_SOFTWARE_ENABLE_DISABLE".DISABLE_FIXTURE.SW_UNIT_02_FIX_2_3_ENABLED AND "DB7300_INTERLOCK_GENERAL".GENERAL_MACHINE.FROM_CELL_TO_MACHINE_GENERAL.CELL_COOLING_DEGRADED_MODE) OR ("DB7300_INTERLOCK_GENERAL".AUX_SIGNALS_INTERFACE.GENERAL."DEGRADED MODE FAULT" AND NOT "DB2120_MPP_ITC_IPC".RESET_FAULTS);
   "DB426_ALARMS_WARNINGS".GENERAL."704401" := "DB7300_INTERLOCK_GENERAL".AUX_SIGNALS_INTERFACE.GENERAL."DEGRADED MODE FAULT";
END_REGION

REGION Network 78: IMMEDIATE STOP ALARMS
   RUNG wire#powerrail
      I_Contact( "DB7300_INTERLOCK_GENERAL".AUX_SIGNALS_INTERFACE.UNIT_01.EMERGENCY_STOP_ACTIVE )
      I_Contact( "DB7300_INTERLOCK_GENERAL".AUX_SIGNALS_INTERFACE.UNIT_01.LIFE_BIT_FAULT )
      I_Contact( "DB7300_INTERLOCK_GENERAL".AUX_SIGNALS_INTERFACE.UNIT_02.EMERGENCY_STOP_ACTIVE )
      I_Contact( "DB7300_INTERLOCK_GENERAL".AUX_SIGNALS_INTERFACE.UNIT_02.LIFE_BIT_FAULT )
      I_Contact( "DB7300_INTERLOCK_GENERAL".AUX_SIGNALS_INTERFACE.GENERAL."DEGRADED MODE FAULT" )
      Not()
      Contact( "M_DUMMY_OFF" )
      { S7_GenerateENO := "TRUE" } Move(in := #FC_NUMBER, out1 => "DB440_MACHINE_ALARM_DECODING".GLOBAL_ALARMS_MACHINE.ALARM_DECODING)
      S_Coil( "DB440_MACHINE_ALARM_DECODING".ALARMS_CENTRAL.IS_ALARMS )
   END_RUNG
   // the same network as SCL:
   // ENO of a box is taken as its EN; it also drops when the box reports an error
   IF NOT (NOT "DB7300_INTERLOCK_GENERAL".AUX_SIGNALS_INTERFACE.UNIT_01.EMERGENCY_STOP_ACTIVE AND NOT "DB7300_INTERLOCK_GENERAL".AUX_SIGNALS_INTERFACE.UNIT_01.LIFE_BIT_FAULT AND NOT "DB7300_INTERLOCK_GENERAL".AUX_SIGNALS_INTERFACE.UNIT_02.EMERGENCY_STOP_ACTIVE AND NOT "DB7300_INTERLOCK_GENERAL".AUX_SIGNALS_INTERFACE.UNIT_02.LIFE_BIT_FAULT AND NOT "DB7300_INTERLOCK_GENERAL".AUX_SIGNALS_INTERFACE.GENERAL."DEGRADED MODE FAULT") AND "M_DUMMY_OFF" THEN
       "DB440_MACHINE_ALARM_DECODING".GLOBAL_ALARMS_MACHINE.ALARM_DECODING := #FC_NUMBER;
       "DB440_MACHINE_ALARM_DECODING".ALARMS_CENTRAL.IS_ALARMS := TRUE;
   END_IF;
END_REGION

REGION Network 79: INMEDIATE STOP AND STOP END OF CYCLE ALARMS
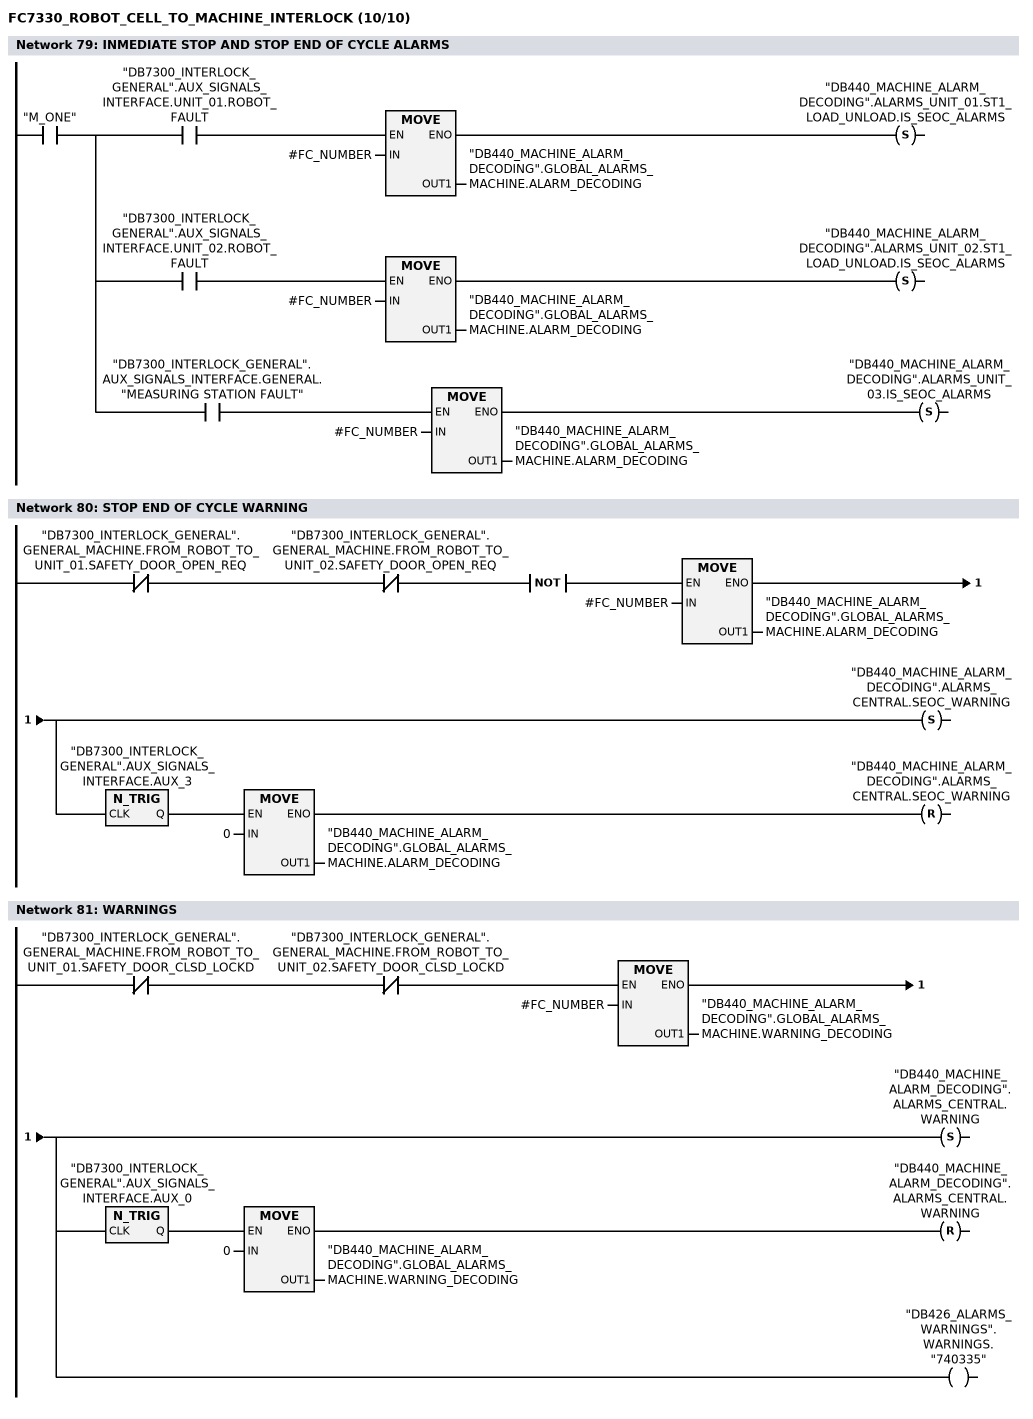
   RUNG wire#powerrail
      Contact( "M_ONE" )
      wire#w1
      Contact( "DB7300_INTERLOCK_GENERAL".AUX_SIGNALS_INTERFACE.UNIT_01.ROBOT_FAULT )
      { S7_GenerateENO := "TRUE" } Move(in := #FC_NUMBER, out1 => "DB440_MACHINE_ALARM_DECODING".GLOBAL_ALARMS_MACHINE.ALARM_DECODING)
      S_Coil( "DB440_MACHINE_ALARM_DECODING".ALARMS_UNIT_01.ST1_LOAD_UNLOAD.IS_SEOC_ALARMS )
   END_RUNG
   RUNG wire#w1
      Contact( "DB7300_INTERLOCK_GENERAL".AUX_SIGNALS_INTERFACE.UNIT_02.ROBOT_FAULT )
      { S7_GenerateENO := "TRUE" } Move(in := #FC_NUMBER, out1 => "DB440_MACHINE_ALARM_DECODING".GLOBAL_ALARMS_MACHINE.ALARM_DECODING)
      S_Coil( "DB440_MACHINE_ALARM_DECODING".ALARMS_UNIT_02.ST1_LOAD_UNLOAD.IS_SEOC_ALARMS )
   END_RUNG
   RUNG wire#w1
      Contact( "DB7300_INTERLOCK_GENERAL".AUX_SIGNALS_INTERFACE.GENERAL."MEASURING STATION FAULT" )
      { S7_GenerateENO := "TRUE" } Move(in := #FC_NUMBER, out1 => "DB440_MACHINE_ALARM_DECODING".GLOBAL_ALARMS_MACHINE.ALARM_DECODING)
      S_Coil( "DB440_MACHINE_ALARM_DECODING".ALARMS_UNIT_03.IS_SEOC_ALARMS )
   END_RUNG
   // the same network as SCL:
   // ENO of a box is taken as its EN; it also drops when the box reports an error
   IF "M_ONE" AND "DB7300_INTERLOCK_GENERAL".AUX_SIGNALS_INTERFACE.UNIT_01.ROBOT_FAULT THEN
       "DB440_MACHINE_ALARM_DECODING".GLOBAL_ALARMS_MACHINE.ALARM_DECODING := #FC_NUMBER;
       "DB440_MACHINE_ALARM_DECODING".ALARMS_UNIT_01.ST1_LOAD_UNLOAD.IS_SEOC_ALARMS := TRUE;
   END_IF;
   IF "M_ONE" AND "DB7300_INTERLOCK_GENERAL".AUX_SIGNALS_INTERFACE.UNIT_02.ROBOT_FAULT THEN
       "DB440_MACHINE_ALARM_DECODING".GLOBAL_ALARMS_MACHINE.ALARM_DECODING := #FC_NUMBER;
       "DB440_MACHINE_ALARM_DECODING".ALARMS_UNIT_02.ST1_LOAD_UNLOAD.IS_SEOC_ALARMS := TRUE;
   END_IF;
   IF "M_ONE" AND "DB7300_INTERLOCK_GENERAL".AUX_SIGNALS_INTERFACE.GENERAL."MEASURING STATION FAULT" THEN
       "DB440_MACHINE_ALARM_DECODING".GLOBAL_ALARMS_MACHINE.ALARM_DECODING := #FC_NUMBER;
       "DB440_MACHINE_ALARM_DECODING".ALARMS_UNIT_03.IS_SEOC_ALARMS := TRUE;
   END_IF;
END_REGION

REGION Network 80: STOP END OF CYCLE WARNING
   RUNG wire#powerrail
      I_Contact( "DB7300_INTERLOCK_GENERAL".GENERAL_MACHINE.FROM_ROBOT_TO_UNIT_01.SAFETY_DOOR_OPEN_REQ )
      I_Contact( "DB7300_INTERLOCK_GENERAL".GENERAL_MACHINE.FROM_ROBOT_TO_UNIT_02.SAFETY_DOOR_OPEN_REQ )
      Not()
      { S7_GenerateENO := "TRUE" } Move(in := #FC_NUMBER, out1 => "DB440_MACHINE_ALARM_DECODING".GLOBAL_ALARMS_MACHINE.ALARM_DECODING)
      wire#w1
      S_Coil( "DB440_MACHINE_ALARM_DECODING".ALARMS_CENTRAL.SEOC_WARNING )
   END_RUNG
   RUNG wire#w1
      N_Trig( "DB7300_INTERLOCK_GENERAL".AUX_SIGNALS_INTERFACE.AUX_3 )
      { S7_GenerateENO := "TRUE" } Move(in := 0, out1 => "DB440_MACHINE_ALARM_DECODING".GLOBAL_ALARMS_MACHINE.ALARM_DECODING)
      R_Coil( "DB440_MACHINE_ALARM_DECODING".ALARMS_CENTRAL.SEOC_WARNING )
   END_RUNG
   // the same network as SCL:
   // ENO of a box is taken as its EN; it also drops when the box reports an error
   #_w1 := NOT (NOT "DB7300_INTERLOCK_GENERAL".GENERAL_MACHINE.FROM_ROBOT_TO_UNIT_01.SAFETY_DOOR_OPEN_REQ AND NOT "DB7300_INTERLOCK_GENERAL".GENERAL_MACHINE.FROM_ROBOT_TO_UNIT_02.SAFETY_DOOR_OPEN_REQ);
   IF #_w1 THEN
       "DB440_MACHINE_ALARM_DECODING".GLOBAL_ALARMS_MACHINE.ALARM_DECODING := #FC_NUMBER;
       "DB440_MACHINE_ALARM_DECODING".ALARMS_CENTRAL.SEOC_WARNING := TRUE;
   END_IF;
   #_w2 := NOT #_w1 AND "DB7300_INTERLOCK_GENERAL".AUX_SIGNALS_INTERFACE.AUX_3;   // falling edge
   "DB7300_INTERLOCK_GENERAL".AUX_SIGNALS_INTERFACE.AUX_3 := #_w1;
   IF #_w2 THEN
       "DB440_MACHINE_ALARM_DECODING".GLOBAL_ALARMS_MACHINE.ALARM_DECODING := 0;
       "DB440_MACHINE_ALARM_DECODING".ALARMS_CENTRAL.SEOC_WARNING := FALSE;
   END_IF;
END_REGION

REGION Network 81: WARNINGS
   RUNG wire#powerrail
      I_Contact( "DB7300_INTERLOCK_GENERAL".GENERAL_MACHINE.FROM_ROBOT_TO_UNIT_01.SAFETY_DOOR_CLSD_LOCKD )
      I_Contact( "DB7300_INTERLOCK_GENERAL".GENERAL_MACHINE.FROM_ROBOT_TO_UNIT_02.SAFETY_DOOR_CLSD_LOCKD )
      Move(in := #FC_NUMBER, out1 => "DB440_MACHINE_ALARM_DECODING".GLOBAL_ALARMS_MACHINE.WARNING_DECODING)
      wire#w1
      S_Coil( "DB440_MACHINE_ALARM_DECODING".ALARMS_CENTRAL.WARNING )
   END_RUNG
   RUNG wire#w1
      N_Trig( "DB7300_INTERLOCK_GENERAL".AUX_SIGNALS_INTERFACE.AUX_0 )
      Move(in := 0, out1 => "DB440_MACHINE_ALARM_DECODING".GLOBAL_ALARMS_MACHINE.WARNING_DECODING)
      R_Coil( "DB440_MACHINE_ALARM_DECODING".ALARMS_CENTRAL.WARNING )
   END_RUNG
   RUNG wire#w1
      Coil( "DB426_ALARMS_WARNINGS".WARNINGS."740335" )
   END_RUNG
   // the same network as SCL:
   #_w1 := NOT "DB7300_INTERLOCK_GENERAL".GENERAL_MACHINE.FROM_ROBOT_TO_UNIT_01.SAFETY_DOOR_CLSD_LOCKD AND NOT "DB7300_INTERLOCK_GENERAL".GENERAL_MACHINE.FROM_ROBOT_TO_UNIT_02.SAFETY_DOOR_CLSD_LOCKD;
   IF #_w1 THEN
       "DB440_MACHINE_ALARM_DECODING".GLOBAL_ALARMS_MACHINE.WARNING_DECODING := #FC_NUMBER;
       "DB440_MACHINE_ALARM_DECODING".ALARMS_CENTRAL.WARNING := TRUE;
   END_IF;
   #_w2 := NOT #_w1 AND "DB7300_INTERLOCK_GENERAL".AUX_SIGNALS_INTERFACE.AUX_0;   // falling edge
   "DB7300_INTERLOCK_GENERAL".AUX_SIGNALS_INTERFACE.AUX_0 := #_w1;
   IF #_w2 THEN
       "DB440_MACHINE_ALARM_DECODING".GLOBAL_ALARMS_MACHINE.WARNING_DECODING := 0;
       "DB440_MACHINE_ALARM_DECODING".ALARMS_CENTRAL.WARNING := FALSE;
   END_IF;
   "DB426_ALARMS_WARNINGS".WARNINGS."740335" := #_w1;
END_REGION
END_FUNCTION
